KUKA KRL program: f1_Kuka_APT201T02S01.SRC

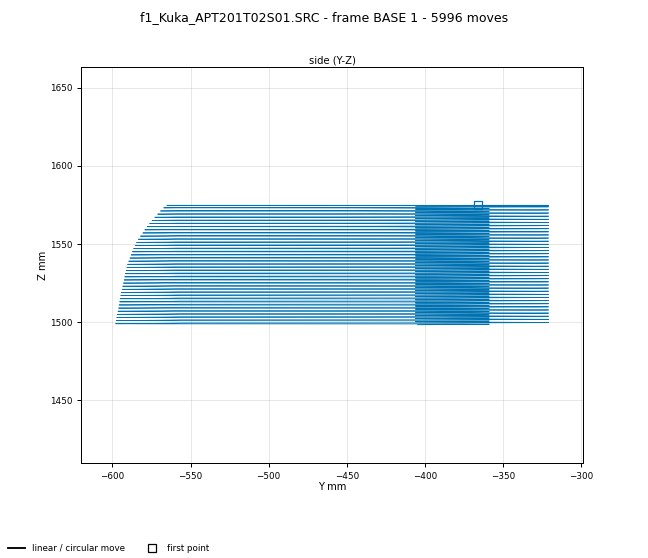
[picture p0: tool path of f1_Kuka_APT201T02S01.SRC in frame BASE 1, 5996 of 5998 moves have a stored position in this frame; points joined in program order, loops and branches not executed]
&ACCESS RVP
&REL 2
&PARAM TEMPLATE = C:\KRC\Roboter\Template\vorgabe
&PARAM EDITMASK = *
DEF f1_Kuka_APT201T02S01()


;FOLD INI;%{PE}%V3.2.0,%MKUKATPBASIS,%CINIT,%VCOMMON,%P
  ;FOLD BAS INI;%{E}%V3.2.0,%MKUKATPBASIS,%CINIT,%VINIT,%P
    GLOBAL INTERRUPT DECL 3 WHEN $STOPMESS==TRUE DO IR_STOPM ( )
    INTERRUPT ON 3
    BAS (#INITMOV,0 )
  ;ENDFOLD (BAS INI)
  ;FOLD USER INI;%{E}%V3.2.0,%MKUKATPUSER,%CINIT,%VINIT,%P
    ;Make your modifications here
  ;ENDFOLD (USER INI)
;ENDFOLD (INI)



;*** Make Initial Position Move
;FOLD PTP PPI1  Vel= 100 % PDAT1 Tool[0] Base[0];%{PE}%R 5.2.22,%MKUKATPBASIS,%CMOVE,%VPTP,%P 1:PTP, 2:PPI1, 3:, 5:100, 7:PDAT1
  $BWDSTART = FALSE
  PDAT_ACT = PPDAT1
  FDAT_ACT = FPPI1
  BAS(#PTP_PARAMS,100)
  PTP XPPI1
;ENDFOLD


;*** Auto Load the Correct TOOL and OFFSET
  ToolChange(2,1)


;*** Make Initial Position Move
;FOLD PTP PPI1  Vel= 100 % PDAT1 Tool[0] Base[0];%{PE}%R 5.2.22,%MKUKATPBASIS,%CMOVE,%VPTP,%P 1:PTP, 2:PPI1, 3:, 5:100, 7:PDAT1
  $BWDSTART = FALSE
  PDAT_ACT = PPDAT1
  FDAT_ACT = FPPI1
  BAS(#PTP_PARAMS,100)
  PTP XPPI1
;ENDFOLD

;*** Auto Load The Correct TOOL Data
  $tool=tool_data[2]

;*** Auto Load The Correct BASE Data
  $base=base_data[1]

  $ADVANCE = 5

SetRPM(8000)

MMPM(30000.0)
LIN {X 0.000,Y -365.799,Z 1574.800,A 0.000,B 0.000,C 90.000,E1 360.000} C_DIS
MMPM(15000.0)
LIN {X 0.000,Y -360.799,Z 1574.800,A 0.000,B 0.000,C 90.000,E1 360.000} C_DIS
MMPM(30000.0)
LIN {X -0.053,Y -359.426,Z 1574.800,A 0.000,B 0.000,C 90.000,E1 354.546} C_DIS
LIN {X 0.070,Y -358.890,Z 1574.800,A 0.000,B 0.000,C 90.000,E1 352.648} C_DIS
LIN {X -0.020,Y -359.563,Z 1574.800,A 0.000,B 0.000,C 90.000,E1 346.645} C_DIS
LIN {X 0.001,Y -361.801,Z 1574.800,A 0.000,B 0.000,C 90.000,E1 339.135} C_DIS
LIN {X -0.154,Y -362.053,Z 1574.800,A 0.000,B 0.000,C 90.000,E1 338.411} C_DIS
LIN {X 0.188,Y -365.979,Z 1574.800,A 0.000,B 0.000,C 90.000,E1 331.641} C_DIS
LIN {X 0.029,Y -366.387,Z 1574.800,A 0.000,B 0.000,C 90.000,E1 330.923} C_DIS
LIN {X -0.031,Y -371.355,Z 1574.800,A 0.000,B 0.000,C 90.000,E1 324.642} C_DIS
LIN {X -0.043,Y -371.766,Z 1574.800,A 0.000,B 0.000,C 90.000,E1 324.276} C_DIS
LIN {X 0.013,Y -377.358,Z 1574.800,A 0.000,B 0.000,C 90.000,E1 318.038} C_DIS
LIN {X 0.012,Y -378.235,Z 1574.800,A 0.000,B 0.000,C 90.000,E1 317.310} C_DIS
LIN {X 0.002,Y -383.940,Z 1574.800,A 0.000,B 0.000,C 90.000,E1 311.515} C_DIS
LIN {X 0.088,Y -384.893,Z 1574.800,A 0.000,B 0.000,C 90.000,E1 310.782} C_DIS
LIN {X 0.262,Y -390.610,Z 1574.800,A 0.000,B 0.000,C 90.000,E1 305.025} C_DIS
LIN {X 0.106,Y -391.104,Z 1574.800,A 0.000,B 0.000,C 90.000,E1 304.692} C_DIS
LIN {X 0.022,Y -391.648,Z 1574.800,A 0.000,B 0.000,C 90.000,E1 303.992} C_DIS
LIN {X -0.080,Y -396.825,Z 1574.800,A 0.000,B 0.000,C 90.000,E1 298.693} C_DIS
LIN {X -0.210,Y -397.120,Z 1574.800,A 0.000,B 0.000,C 90.000,E1 298.359} C_DIS
LIN {X -0.055,Y -401.597,Z 1574.800,A 0.000,B 0.000,C 90.000,E1 292.717} C_DIS
LIN {X 0.221,Y -404.659,Z 1574.800,A 0.000,B 0.000,C 90.000,E1 287.094} C_DIS
LIN {X -0.079,Y -404.735,Z 1574.800,A 0.000,B 0.000,C 90.000,E1 286.441} C_DIS
LIN {X 0.214,Y -406.099,Z 1574.800,A 0.000,B 0.000,C 90.000,E1 281.535} C_DIS
LIN {X -0.176,Y -406.094,Z 1574.800,A 0.000,B 0.000,C 90.000,E1 281.243} C_DIS
LIN {X -0.098,Y -405.680,Z 1574.800,A 0.000,B 0.000,C 90.000,E1 276.024} C_DIS
LIN {X -0.165,Y -405.058,Z 1574.800,A 0.000,B 0.000,C 90.000,E1 274.992} C_DIS
LIN {X -0.060,Y -403.497,Z 1574.800,A 0.000,B 0.000,C 90.000,E1 270.802} C_DIS
LIN {X -0.092,Y -403.288,Z 1574.800,A 0.000,B 0.000,C 90.000,E1 270.458} C_DIS
LIN {X 0.091,Y -398.931,Z 1574.800,A 0.000,B 0.000,C 90.000,E1 264.837} C_DIS
LIN {X -0.040,Y -393.108,Z 1574.800,A 0.000,B 0.000,C 90.000,E1 259.567} C_DIS
LIN {X -0.080,Y -392.836,Z 1574.800,A 0.000,B 0.000,C 90.000,E1 259.218} C_DIS
LIN {X 0.034,Y -385.993,Z 1574.800,A 0.000,B 0.000,C 90.000,E1 254.212} C_DIS
LIN {X -0.026,Y -385.267,Z 1574.800,A 0.000,B 0.000,C 90.000,E1 253.504} C_DIS
LIN {X -0.004,Y -384.767,Z 1574.800,A 0.000,B 0.000,C 90.000,E1 253.142} C_DIS
LIN {X 0.220,Y -377.972,Z 1574.800,A 0.000,B 0.000,C 90.000,E1 248.773} C_DIS
LIN {X -0.044,Y -376.233,Z 1574.800,A 0.000,B 0.000,C 90.000,E1 247.358} C_DIS
LIN {X 0.057,Y -374.944,Z 1574.800,A 0.000,B 0.000,C 90.000,E1 246.613} C_DIS
LIN {X -0.208,Y -368.417,Z 1574.800,A 0.000,B 0.000,C 90.000,E1 242.615} C_DIS
LIN {X 0.097,Y -366.047,Z 1574.800,A 0.000,B 0.000,C 90.000,E1 240.717} C_DIS
LIN {X 0.004,Y -359.196,Z 1574.800,A 0.000,B 0.000,C 90.000,E1 236.628} C_DIS
LIN {X 0.021,Y -355.842,Z 1574.800,A 0.000,B 0.000,C 90.000,E1 233.989} C_DIS
LIN {X -0.173,Y -348.793,Z 1574.800,A 0.000,B 0.000,C 90.000,E1 229.461} C_DIS
LIN {X -0.097,Y -346.185,Z 1574.800,A 0.000,B 0.000,C 90.000,E1 227.148} C_DIS
LIN {X -0.089,Y -345.065,Z 1574.800,A 0.000,B 0.000,C 90.000,E1 226.377} C_DIS
LIN {X 0.094,Y -338.586,Z 1574.800,A 0.000,B 0.000,C 90.000,E1 221.310} C_DIS
LIN {X 0.094,Y -336.840,Z 1574.800,A 0.000,B 0.000,C 90.000,E1 219.358} C_DIS
LIN {X 0.014,Y -330.861,Z 1574.800,A 0.000,B 0.000,C 90.000,E1 213.865} C_DIS
LIN {X 0.149,Y -329.296,Z 1574.800,A 0.000,B 0.000,C 90.000,E1 211.465} C_DIS
LIN {X -0.154,Y -324.669,Z 1574.800,A 0.000,B 0.000,C 90.000,E1 205.540} C_DIS
LIN {X 0.174,Y -323.838,Z 1574.800,A 0.000,B 0.000,C 90.000,E1 203.078} C_DIS
LIN {X -0.018,Y -321.123,Z 1574.800,A 0.000,B 0.000,C 90.000,E1 194.662} C_DIS
LIN {X 0.138,Y -320.932,Z 1574.800,A 0.000,B 0.000,C 90.000,E1 193.828} C_DIS
LIN {X -0.076,Y -321.563,Z 1574.800,A 0.000,B 0.000,C 90.000,E1 185.796} C_DIS
LIN {X -0.143,Y -324.415,Z 1574.800,A 0.000,B 0.000,C 90.000,E1 178.165} C_DIS
LIN {X -0.141,Y -325.376,Z 1574.800,A 0.000,B 0.000,C 90.000,E1 176.963} C_DIS
LIN {X -0.100,Y -329.112,Z 1574.800,A 0.000,B 0.000,C 90.000,E1 170.971} C_DIS
LIN {X 0.061,Y -334.260,Z 1574.800,A 0.000,B 0.000,C 90.000,E1 166.589} C_DIS
LIN {X 0.067,Y -335.488,Z 1574.800,A 0.000,B 0.000,C 90.000,E1 165.408} C_DIS
LIN {X 0.143,Y -340.932,Z 1574.800,A 0.000,B 0.000,C 90.000,E1 161.094} C_DIS
LIN {X -0.172,Y -342.138,Z 1574.800,A 0.000,B 0.000,C 90.000,E1 160.369} C_DIS
LIN {X -0.058,Y -347.939,Z 1574.800,A 0.000,B 0.000,C 90.000,E1 156.102} C_DIS
LIN {X -0.082,Y -354.260,Z 1574.800,A 0.000,B 0.000,C 90.000,E1 152.666} C_DIS
LIN {X -0.222,Y -361.406,Z 1574.800,A 0.000,B 0.000,C 90.000,E1 148.535} C_DIS
LIN {X 0.064,Y -368.758,Z 1574.800,A 0.000,B 0.000,C 90.000,E1 145.135} C_DIS
LIN {X 0.064,Y -377.030,Z 1574.800,A 0.000,B 0.000,C 90.000,E1 141.090} C_DIS
LIN {X -0.061,Y -383.435,Z 1574.800,A 0.000,B 0.000,C 90.000,E1 138.566} C_DIS
LIN {X -0.015,Y -385.037,Z 1574.800,A 0.000,B 0.000,C 90.000,E1 137.838} C_DIS
LIN {X -0.004,Y -394.325,Z 1574.800,A 0.000,B 0.000,C 90.000,E1 133.905} C_DIS
LIN {X 0.107,Y -399.276,Z 1574.800,A 0.000,B 0.000,C 90.000,E1 132.123} C_DIS
LIN {X 0.210,Y -400.192,Z 1574.800,A 0.000,B 0.000,C 90.000,E1 131.757} C_DIS
LIN {X -0.113,Y -409.687,Z 1574.800,A 0.000,B 0.000,C 90.000,E1 127.971} C_DIS
LIN {X 0.046,Y -415.746,Z 1574.800,A 0.000,B 0.000,C 90.000,E1 125.884} C_DIS
LIN {X 0.152,Y -425.188,Z 1574.800,A 0.000,B 0.000,C 90.000,E1 122.133} C_DIS
LIN {X 0.086,Y -430.187,Z 1574.800,A 0.000,B 0.000,C 90.000,E1 120.463} C_DIS
LIN {X 0.085,Y -431.108,Z 1574.800,A 0.000,B 0.000,C 90.000,E1 120.129} C_DIS
LIN {X 0.032,Y -440.206,Z 1574.800,A 0.000,B 0.000,C 90.000,E1 116.488} C_DIS
LIN {X 0.039,Y -444.962,Z 1574.800,A 0.000,B 0.000,C 90.000,E1 114.847} C_DIS
LIN {X -0.108,Y -454.089,Z 1574.800,A 0.000,B 0.000,C 90.000,E1 110.972} C_DIS
LIN {X 0.003,Y -456.743,Z 1574.800,A 0.000,B 0.000,C 90.000,E1 109.993} C_DIS
LIN {X -0.096,Y -457.517,Z 1574.800,A 0.000,B 0.000,C 90.000,E1 109.685} C_DIS
LIN {X -0.150,Y -466.200,Z 1574.800,A 0.000,B 0.000,C 90.000,E1 105.552} C_DIS
LIN {X 0.026,Y -467.764,Z 1574.800,A 0.000,B 0.000,C 90.000,E1 104.898} C_DIS
LIN {X -0.209,Y -469.313,Z 1574.800,A 0.000,B 0.000,C 90.000,E1 103.883} C_DIS
LIN {X 0.252,Y -548.916,Z 1574.800,A 0.000,B 0.000,C 90.000,E1 103.828} C_DIS
LIN {X -0.055,Y -550.377,Z 1574.800,A 0.000,B 0.000,C 90.000,E1 103.647} C_DIS
LIN {X 0.049,Y -551.250,Z 1574.800,A 0.000,B 0.000,C 90.000,E1 103.355} C_DIS
LIN {X -0.263,Y -552.432,Z 1574.800,A 0.000,B 0.000,C 90.000,E1 102.827} C_DIS
LIN {X 0.096,Y -553.523,Z 1574.800,A 0.000,B 0.000,C 90.000,E1 101.951} C_DIS
LIN {X -0.073,Y -554.401,Z 1574.800,A 0.000,B 0.000,C 90.000,E1 101.130} C_DIS
LIN {X -0.236,Y -555.112,Z 1574.800,A 0.000,B 0.000,C 90.000,E1 100.310} C_DIS
LIN {X -0.102,Y -556.191,Z 1574.800,A 0.000,B 0.000,C 90.000,E1 98.624} C_DIS
LIN {X -0.289,Y -556.849,Z 1574.800,A 0.000,B 0.000,C 90.000,E1 97.530} C_DIS
LIN {X -0.203,Y -557.535,Z 1574.800,A 0.000,B 0.000,C 90.000,E1 95.853} C_DIS
LIN {X -0.219,Y -557.914,Z 1574.800,A 0.000,B 0.000,C 90.000,E1 94.188} C_DIS
LIN {X -0.221,Y -558.368,Z 1574.800,A 0.000,B 0.000,C 90.000,E1 92.522} C_DIS
LIN {X 0.226,Y -558.750,Z 1574.800,A 0.000,B 0.000,C 90.000,E1 91.088} C_DIS
LIN {X -0.272,Y -559.196,Z 1574.800,A 0.000,B 0.000,C 90.000,E1 89.198} C_DIS
LIN {X -0.191,Y -559.752,Z 1574.800,A 0.000,B 0.000,C 90.000,E1 87.249} C_DIS
LIN {X -0.157,Y -560.343,Z 1574.800,A 0.000,B 0.000,C 90.000,E1 85.584} C_DIS
LIN {X 0.022,Y -561.145,Z 1574.800,A 0.000,B 0.000,C 90.000,E1 83.628} C_DIS
LIN {X -0.132,Y -562.271,Z 1574.800,A 0.000,B 0.000,C 90.000,E1 81.432} C_DIS
LIN {X -0.235,Y -563.276,Z 1574.800,A 0.000,B 0.000,C 90.000,E1 79.511} C_DIS
LIN {X 0.073,Y -564.218,Z 1574.800,A 0.000,B 0.000,C 90.000,E1 77.825} C_DIS
LIN {X 0.080,Y -564.877,Z 1574.800,A 0.000,B 0.000,C 90.000,E1 76.172} C_DIS
LIN {X -0.219,Y -565.104,Z 1574.800,A 0.000,B 0.000,C 90.000,E1 75.102} C_DIS
LIN {X -0.128,Y -565.147,Z 1574.800,A 0.000,B 0.000,C 90.000,E1 74.267} C_DIS
LIN {X 0.121,Y -564.945,Z 1574.800,A 0.000,B 0.000,C 90.000,E1 73.142} C_DIS
LIN {X 0.053,Y -564.549,Z 1574.800,A 0.000,B 0.000,C 90.000,E1 72.598} C_DIS
LIN {X -0.014,Y -563.765,Z 1574.800,A 0.000,B 0.000,C 90.000,E1 72.054} C_DIS
LIN {X -0.167,Y -562.900,Z 1574.800,A 0.000,B 0.000,C 90.000,E1 71.764} C_DIS
LIN {X -0.031,Y -562.209,Z 1574.800,A 0.000,B 0.000,C 90.000,E1 71.638} C_DIS
LIN {X -0.274,Y -561.841,Z 1574.800,A 0.000,B 0.000,C 90.000,E1 71.638} C_DIS
LIN {X 0.177,Y -473.244,Z 1574.800,A 0.000,B 0.000,C 90.000,E1 71.583} C_DIS
LIN {X 0.025,Y -465.713,Z 1574.800,A 0.000,B 0.000,C 90.000,E1 67.102} C_DIS
LIN {X -0.179,Y -456.183,Z 1574.800,A 0.000,B 0.000,C 90.000,E1 62.359} C_DIS
LIN {X -0.073,Y -455.666,Z 1574.800,A 0.000,B 0.000,C 90.000,E1 62.025} C_DIS
LIN {X -0.081,Y -454.178,Z 1574.800,A 0.000,B 0.000,C 90.000,E1 61.385} C_DIS
LIN {X 0.021,Y -445.148,Z 1574.800,A 0.000,B 0.000,C 90.000,E1 57.168} C_DIS
LIN {X 0.146,Y -443.995,Z 1574.800,A 0.000,B 0.000,C 90.000,E1 56.501} C_DIS
LIN {X 0.091,Y -433.537,Z 1574.800,A 0.000,B 0.000,C 90.000,E1 51.904} C_DIS
LIN {X -0.063,Y -431.699,Z 1574.800,A 0.000,B 0.000,C 90.000,E1 50.928} C_DIS
LIN {X 0.096,Y -429.255,Z 1574.800,A 0.000,B 0.000,C 90.000,E1 49.908} C_DIS
LIN {X -0.126,Y -419.923,Z 1574.800,A 0.000,B 0.000,C 90.000,E1 45.567} C_DIS
LIN {X -0.048,Y -418.732,Z 1574.800,A 0.000,B 0.000,C 90.000,E1 44.879} C_DIS
LIN {X -0.082,Y -409.803,Z 1574.800,A 0.000,B 0.000,C 90.000,E1 40.782} C_DIS
LIN {X -0.045,Y -406.207,Z 1574.800,A 0.000,B 0.000,C 90.000,E1 38.705} C_DIS
LIN {X 0.100,Y -405.567,Z 1574.800,A 0.000,B 0.000,C 90.000,E1 38.338} C_DIS
LIN {X 0.175,Y -396.741,Z 1574.800,A 0.000,B 0.000,C 90.000,E1 33.785} C_DIS
LIN {X 0.155,Y -393.529,Z 1574.800,A 0.000,B 0.000,C 90.000,E1 31.671} C_DIS
LIN {X -0.093,Y -386.172,Z 1574.800,A 0.000,B 0.000,C 90.000,E1 27.436} C_DIS
LIN {X 0.055,Y -382.972,Z 1574.800,A 0.000,B 0.000,C 90.000,E1 24.899} C_DIS
LIN {X 0.036,Y -376.689,Z 1574.800,A 0.000,B 0.000,C 90.000,E1 20.556} C_DIS
LIN {X 0.019,Y -373.753,Z 1574.800,A 0.000,B 0.000,C 90.000,E1 17.638} C_DIS
LIN {X -0.034,Y -372.850,Z 1574.800,A 0.000,B 0.000,C 90.000,E1 16.913} C_DIS
LIN {X -0.131,Y -367.590,Z 1574.800,A 0.000,B 0.000,C 90.000,E1 11.771} C_DIS
LIN {X -0.047,Y -366.471,Z 1574.800,A 0.000,B 0.000,C 90.000,E1 9.905} C_DIS
LIN {X -0.109,Y -361.776,Z 1574.800,A 0.000,B 0.000,C 90.000,E1 3.955} C_DIS
LIN {X 0.136,Y -360.896,Z 1574.800,A 0.000,B 0.000,C 90.000,E1 0.172} C_DIS
LIN {X -0.053,Y -359.426,Z 1574.770,A 0.000,B 0.000,C 90.000,E1 354.546} C_DIS
LIN {X 0.070,Y -358.890,Z 1574.759,A 0.000,B 0.000,C 90.000,E1 352.648} C_DIS
LIN {X -0.020,Y -359.563,Z 1574.726,A 0.000,B 0.000,C 90.000,E1 346.645} C_DIS
LIN {X 0.001,Y -361.801,Z 1574.684,A 0.000,B 0.000,C 90.000,E1 339.135} C_DIS
LIN {X -0.154,Y -362.053,Z 1574.680,A 0.000,B 0.000,C 90.000,E1 338.411} C_DIS
LIN {X 0.189,Y -365.980,Z 1574.643,A 0.000,B 0.000,C 90.000,E1 331.641} C_DIS
LIN {X 0.029,Y -366.387,Z 1574.639,A 0.000,B 0.000,C 90.000,E1 330.923} C_DIS
LIN {X -0.031,Y -371.355,Z 1574.604,A 0.000,B 0.000,C 90.000,E1 324.642} C_DIS
LIN {X -0.043,Y -371.766,Z 1574.602,A 0.000,B 0.000,C 90.000,E1 324.276} C_DIS
LIN {X 0.013,Y -377.358,Z 1574.567,A 0.000,B 0.000,C 90.000,E1 318.038} C_DIS
LIN {X 0.012,Y -378.235,Z 1574.563,A 0.000,B 0.000,C 90.000,E1 317.310} C_DIS
LIN {X 0.002,Y -383.940,Z 1574.531,A 0.000,B 0.000,C 90.000,E1 311.515} C_DIS
LIN {X 0.088,Y -384.893,Z 1574.527,A 0.000,B 0.000,C 90.000,E1 310.782} C_DIS
LIN {X 0.262,Y -390.610,Z 1574.495,A 0.000,B 0.000,C 90.000,E1 305.025} C_DIS
LIN {X 0.106,Y -391.104,Z 1574.493,A 0.000,B 0.000,C 90.000,E1 304.692} C_DIS
LIN {X 0.022,Y -391.648,Z 1574.489,A 0.000,B 0.000,C 90.000,E1 303.992} C_DIS
LIN {X -0.080,Y -396.825,Z 1574.459,A 0.000,B 0.000,C 90.000,E1 298.693} C_DIS
LIN {X -0.210,Y -397.120,Z 1574.457,A 0.000,B 0.000,C 90.000,E1 298.359} C_DIS
LIN {X -0.055,Y -401.597,Z 1574.426,A 0.000,B 0.000,C 90.000,E1 292.717} C_DIS
LIN {X 0.222,Y -404.659,Z 1574.395,A 0.000,B 0.000,C 90.000,E1 287.094} C_DIS
LIN {X -0.079,Y -404.735,Z 1574.391,A 0.000,B 0.000,C 90.000,E1 286.441} C_DIS
LIN {X 0.214,Y -406.099,Z 1574.364,A 0.000,B 0.000,C 90.000,E1 281.535} C_DIS
LIN {X -0.176,Y -406.094,Z 1574.362,A 0.000,B 0.000,C 90.000,E1 281.243} C_DIS
LIN {X -0.097,Y -405.680,Z 1574.333,A 0.000,B 0.000,C 90.000,E1 276.024} C_DIS
LIN {X -0.165,Y -405.058,Z 1574.328,A 0.000,B 0.000,C 90.000,E1 274.992} C_DIS
LIN {X -0.060,Y -403.497,Z 1574.304,A 0.000,B 0.000,C 90.000,E1 270.802} C_DIS
LIN {X -0.092,Y -403.288,Z 1574.302,A 0.000,B 0.000,C 90.000,E1 270.458} C_DIS
LIN {X 0.091,Y -398.931,Z 1574.271,A 0.000,B 0.000,C 90.000,E1 264.837} C_DIS
LIN {X -0.040,Y -393.108,Z 1574.242,A 0.000,B 0.000,C 90.000,E1 259.567} C_DIS
LIN {X -0.079,Y -392.835,Z 1574.240,A 0.000,B 0.000,C 90.000,E1 259.218} C_DIS
LIN {X 0.034,Y -385.993,Z 1574.212,A 0.000,B 0.000,C 90.000,E1 254.212} C_DIS
LIN {X -0.026,Y -385.267,Z 1574.208,A 0.000,B 0.000,C 90.000,E1 253.504} C_DIS
LIN {X -0.004,Y -384.768,Z 1574.206,A 0.000,B 0.000,C 90.000,E1 253.142} C_DIS
LIN {X 0.221,Y -377.973,Z 1574.182,A 0.000,B 0.000,C 90.000,E1 248.773} C_DIS
LIN {X -0.044,Y -376.233,Z 1574.174,A 0.000,B 0.000,C 90.000,E1 247.358} C_DIS
LIN {X 0.057,Y -374.944,Z 1574.170,A 0.000,B 0.000,C 90.000,E1 246.613} C_DIS
LIN {X -0.208,Y -368.417,Z 1574.148,A 0.000,B 0.000,C 90.000,E1 242.615} C_DIS
LIN {X 0.097,Y -366.047,Z 1574.137,A 0.000,B 0.000,C 90.000,E1 240.717} C_DIS
LIN {X 0.004,Y -359.196,Z 1574.115,A 0.000,B 0.000,C 90.000,E1 236.628} C_DIS
LIN {X 0.021,Y -355.842,Z 1574.100,A 0.000,B 0.000,C 90.000,E1 233.989} C_DIS
LIN {X -0.173,Y -348.793,Z 1574.075,A 0.000,B 0.000,C 90.000,E1 229.461} C_DIS
LIN {X -0.097,Y -346.185,Z 1574.062,A 0.000,B 0.000,C 90.000,E1 227.148} C_DIS
LIN {X -0.088,Y -345.065,Z 1574.058,A 0.000,B 0.000,C 90.000,E1 226.377} C_DIS
LIN {X 0.094,Y -338.586,Z 1574.030,A 0.000,B 0.000,C 90.000,E1 221.310} C_DIS
LIN {X 0.094,Y -336.840,Z 1574.019,A 0.000,B 0.000,C 90.000,E1 219.358} C_DIS
LIN {X 0.014,Y -330.861,Z 1573.988,A 0.000,B 0.000,C 90.000,E1 213.865} C_DIS
LIN {X 0.149,Y -329.296,Z 1573.975,A 0.000,B 0.000,C 90.000,E1 211.465} C_DIS
LIN {X -0.154,Y -324.669,Z 1573.942,A 0.000,B 0.000,C 90.000,E1 205.540} C_DIS
LIN {X 0.174,Y -323.837,Z 1573.928,A 0.000,B 0.000,C 90.000,E1 203.078} C_DIS
LIN {X -0.017,Y -321.124,Z 1573.881,A 0.000,B 0.000,C 90.000,E1 194.662} C_DIS
LIN {X 0.138,Y -320.932,Z 1573.877,A 0.000,B 0.000,C 90.000,E1 193.828} C_DIS
LIN {X -0.076,Y -321.562,Z 1573.832,A 0.000,B 0.000,C 90.000,E1 185.796} C_DIS
LIN {X -0.143,Y -324.415,Z 1573.790,A 0.000,B 0.000,C 90.000,E1 178.165} C_DIS
LIN {X -0.141,Y -325.376,Z 1573.783,A 0.000,B 0.000,C 90.000,E1 176.963} C_DIS
LIN {X -0.100,Y -329.112,Z 1573.750,A 0.000,B 0.000,C 90.000,E1 170.971} C_DIS
LIN {X 0.061,Y -334.260,Z 1573.726,A 0.000,B 0.000,C 90.000,E1 166.589} C_DIS
LIN {X 0.067,Y -335.488,Z 1573.719,A 0.000,B 0.000,C 90.000,E1 165.408} C_DIS
LIN {X 0.143,Y -340.932,Z 1573.695,A 0.000,B 0.000,C 90.000,E1 161.094} C_DIS
LIN {X -0.172,Y -342.138,Z 1573.691,A 0.000,B 0.000,C 90.000,E1 160.369} C_DIS
LIN {X -0.058,Y -347.939,Z 1573.667,A 0.000,B 0.000,C 90.000,E1 156.102} C_DIS
LIN {X -0.081,Y -354.259,Z 1573.648,A 0.000,B 0.000,C 90.000,E1 152.666} C_DIS
LIN {X -0.222,Y -361.406,Z 1573.625,A 0.000,B 0.000,C 90.000,E1 148.535} C_DIS
LIN {X 0.065,Y -368.758,Z 1573.606,A 0.000,B 0.000,C 90.000,E1 145.135} C_DIS
LIN {X 0.065,Y -377.029,Z 1573.584,A 0.000,B 0.000,C 90.000,E1 141.090} C_DIS
LIN {X -0.061,Y -383.435,Z 1573.570,A 0.000,B 0.000,C 90.000,E1 138.566} C_DIS
LIN {X -0.015,Y -385.037,Z 1573.566,A 0.000,B 0.000,C 90.000,E1 137.838} C_DIS
LIN {X -0.004,Y -394.325,Z 1573.544,A 0.000,B 0.000,C 90.000,E1 133.905} C_DIS
LIN {X 0.107,Y -399.276,Z 1573.534,A 0.000,B 0.000,C 90.000,E1 132.123} C_DIS
LIN {X 0.210,Y -400.192,Z 1573.532,A 0.000,B 0.000,C 90.000,E1 131.757} C_DIS
LIN {X -0.113,Y -409.687,Z 1573.511,A 0.000,B 0.000,C 90.000,E1 127.971} C_DIS
LIN {X 0.046,Y -415.746,Z 1573.499,A 0.000,B 0.000,C 90.000,E1 125.884} C_DIS
LIN {X 0.153,Y -425.188,Z 1573.479,A 0.000,B 0.000,C 90.000,E1 122.133} C_DIS
LIN {X 0.087,Y -430.186,Z 1573.469,A 0.000,B 0.000,C 90.000,E1 120.463} C_DIS
LIN {X 0.086,Y -431.107,Z 1573.468,A 0.000,B 0.000,C 90.000,E1 120.129} C_DIS
LIN {X 0.032,Y -440.207,Z 1573.447,A 0.000,B 0.000,C 90.000,E1 116.488} C_DIS
LIN {X 0.039,Y -444.962,Z 1573.438,A 0.000,B 0.000,C 90.000,E1 114.847} C_DIS
LIN {X -0.108,Y -454.089,Z 1573.417,A 0.000,B 0.000,C 90.000,E1 110.972} C_DIS
LIN {X 0.005,Y -456.742,Z 1573.411,A 0.000,B 0.000,C 90.000,E1 109.993} C_DIS
LIN {X -0.096,Y -457.517,Z 1573.409,A 0.000,B 0.000,C 90.000,E1 109.685} C_DIS
LIN {X -0.047,Y -465.767,Z 1573.387,A 0.000,B 0.000,C 90.000,E1 105.717} C_DIS
LIN {X -0.088,Y -548.675,Z 1573.387,A 0.000,B 0.000,C 90.000,E1 105.717} C_DIS
LIN {X -0.153,Y -548.982,Z 1573.387,A 0.000,B 0.000,C 90.000,E1 105.717} C_DIS
LIN {X -0.177,Y -550.294,Z 1573.386,A 0.000,B 0.000,C 90.000,E1 105.552} C_DIS
LIN {X 0.069,Y -551.293,Z 1573.385,A 0.000,B 0.000,C 90.000,E1 105.245} C_DIS
LIN {X 0.175,Y -551.975,Z 1573.383,A 0.000,B 0.000,C 90.000,E1 104.954} C_DIS
LIN {X 0.004,Y -552.984,Z 1573.380,A 0.000,B 0.000,C 90.000,E1 104.411} C_DIS
LIN {X 0.239,Y -553.715,Z 1573.377,A 0.000,B 0.000,C 90.000,E1 103.828} C_DIS
LIN {X 0.196,Y -554.850,Z 1573.371,A 0.000,B 0.000,C 90.000,E1 102.715} C_DIS
LIN {X -0.236,Y -555.849,Z 1573.363,A 0.000,B 0.000,C 90.000,E1 101.366} C_DIS
LIN {X -0.248,Y -556.511,Z 1573.357,A 0.000,B 0.000,C 90.000,E1 100.254} C_DIS
LIN {X 0.051,Y -557.419,Z 1573.346,A 0.000,B 0.000,C 90.000,E1 98.276} C_DIS
LIN {X -0.181,Y -557.796,Z 1573.341,A 0.000,B 0.000,C 90.000,E1 97.466} C_DIS
LIN {X -0.147,Y -558.339,Z 1573.332,A 0.000,B 0.000,C 90.000,E1 95.796} C_DIS
LIN {X -0.143,Y -558.609,Z 1573.323,A 0.000,B 0.000,C 90.000,E1 94.131} C_DIS
LIN {X -0.131,Y -558.995,Z 1573.314,A 0.000,B 0.000,C 90.000,E1 92.465} C_DIS
LIN {X -0.230,Y -559.336,Z 1573.306,A 0.000,B 0.000,C 90.000,E1 91.088} C_DIS
LIN {X -0.156,Y -559.756,Z 1573.295,A 0.000,B 0.000,C 90.000,E1 89.141} C_DIS
LIN {X -0.061,Y -560.327,Z 1573.284,A 0.000,B 0.000,C 90.000,E1 87.192} C_DIS
LIN {X -0.015,Y -560.941,Z 1573.275,A 0.000,B 0.000,C 90.000,E1 85.527} C_DIS
LIN {X 0.178,Y -561.807,Z 1573.264,A 0.000,B 0.000,C 90.000,E1 83.571} C_DIS
LIN {X 0.041,Y -563.034,Z 1573.252,A 0.000,B 0.000,C 90.000,E1 81.376} C_DIS
LIN {X -0.044,Y -564.180,Z 1573.241,A 0.000,B 0.000,C 90.000,E1 79.454} C_DIS
LIN {X -0.152,Y -565.281,Z 1573.232,A 0.000,B 0.000,C 90.000,E1 77.813} C_DIS
LIN {X -0.241,Y -566.169,Z 1573.223,A 0.000,B 0.000,C 90.000,E1 76.172} C_DIS
LIN {X 0.192,Y -566.734,Z 1573.215,A 0.000,B 0.000,C 90.000,E1 74.755} C_DIS
LIN {X 0.240,Y -567.099,Z 1573.208,A 0.000,B 0.000,C 90.000,E1 73.378} C_DIS
LIN {X -0.193,Y -567.140,Z 1573.203,A 0.000,B 0.000,C 90.000,E1 72.598} C_DIS
LIN {X 0.244,Y -566.843,Z 1573.197,A 0.000,B 0.000,C 90.000,E1 71.456} C_DIS
LIN {X -0.198,Y -566.323,Z 1573.193,A 0.000,B 0.000,C 90.000,E1 70.678} C_DIS
LIN {X -0.065,Y -565.425,Z 1573.190,A 0.000,B 0.000,C 90.000,E1 70.115} C_DIS
LIN {X -0.069,Y -564.450,Z 1573.188,A 0.000,B 0.000,C 90.000,E1 69.752} C_DIS
LIN {X 0.067,Y -563.822,Z 1573.187,A 0.000,B 0.000,C 90.000,E1 69.625} C_DIS
LIN {X 0.239,Y -563.373,Z 1573.187,A 0.000,B 0.000,C 90.000,E1 69.571} C_DIS
LIN {X 0.182,Y -563.196,Z 1573.187,A 0.000,B 0.000,C 90.000,E1 69.571} C_DIS
LIN {X 0.104,Y -469.466,Z 1573.187,A 0.000,B 0.000,C 90.000,E1 69.571} C_DIS
LIN {X -0.082,Y -465.606,Z 1573.172,A 0.000,B 0.000,C 90.000,E1 67.050} C_DIS
LIN {X -0.203,Y -456.601,Z 1573.148,A 0.000,B 0.000,C 90.000,E1 62.615} C_DIS
LIN {X -0.203,Y -455.561,Z 1573.144,A 0.000,B 0.000,C 90.000,E1 61.975} C_DIS
LIN {X -0.199,Y -445.620,Z 1573.119,A 0.000,B 0.000,C 90.000,E1 57.454} C_DIS
LIN {X 0.233,Y -443.853,Z 1573.114,A 0.000,B 0.000,C 90.000,E1 56.421} C_DIS
LIN {X 0.245,Y -434.703,Z 1573.092,A 0.000,B 0.000,C 90.000,E1 52.477} C_DIS
LIN {X -0.252,Y -431.576,Z 1573.083,A 0.000,B 0.000,C 90.000,E1 50.884} C_DIS
LIN {X -0.044,Y -421.692,Z 1573.058,A 0.000,B 0.000,C 90.000,E1 46.500} C_DIS
LIN {X 0.025,Y -418.597,Z 1573.049,A 0.000,B 0.000,C 90.000,E1 44.798} C_DIS
LIN {X -0.170,Y -409.031,Z 1573.024,A 0.000,B 0.000,C 90.000,E1 40.378} C_DIS
LIN {X 0.012,Y -406.092,Z 1573.015,A 0.000,B 0.000,C 90.000,E1 38.624} C_DIS
LIN {X -0.131,Y -403.868,Z 1573.009,A 0.000,B 0.000,C 90.000,E1 37.604} C_DIS
LIN {X -0.038,Y -395.519,Z 1572.984,A 0.000,B 0.000,C 90.000,E1 33.038} C_DIS
LIN {X -0.218,Y -393.987,Z 1572.978,A 0.000,B 0.000,C 90.000,E1 32.005} C_DIS
LIN {X 0.051,Y -392.679,Z 1572.974,A 0.000,B 0.000,C 90.000,E1 31.258} C_DIS
LIN {X 0.092,Y -385.076,Z 1572.948,A 0.000,B 0.000,C 90.000,E1 26.616} C_DIS
LIN {X 0.060,Y -382.887,Z 1572.938,A 0.000,B 0.000,C 90.000,E1 24.823} C_DIS
LIN {X 0.007,Y -376.178,Z 1572.912,A 0.000,B 0.000,C 90.000,E1 20.120} C_DIS
LIN {X -0.124,Y -373.690,Z 1572.898,A 0.000,B 0.000,C 90.000,E1 17.583} C_DIS
LIN {X 0.011,Y -368.087,Z 1572.869,A 0.000,B 0.000,C 90.000,E1 12.411} C_DIS
LIN {X -0.181,Y -366.407,Z 1572.855,A 0.000,B 0.000,C 90.000,E1 9.849} C_DIS
LIN {X 0.118,Y -361.742,Z 1572.822,A 0.000,B 0.000,C 90.000,E1 3.841} C_DIS
LIN {X 0.004,Y -360.864,Z 1572.801,A 0.000,B 0.000,C 90.000,E1 0.115} C_DIS
LIN {X -0.053,Y -359.426,Z 1572.770,A 0.000,B 0.000,C 90.000,E1 354.546} C_DIS
LIN {X 0.070,Y -358.890,Z 1572.759,A 0.000,B 0.000,C 90.000,E1 352.648} C_DIS
LIN {X -0.020,Y -359.563,Z 1572.726,A 0.000,B 0.000,C 90.000,E1 346.645} C_DIS
LIN {X 0.001,Y -361.801,Z 1572.684,A 0.000,B 0.000,C 90.000,E1 339.135} C_DIS
LIN {X -0.154,Y -362.053,Z 1572.680,A 0.000,B 0.000,C 90.000,E1 338.411} C_DIS
LIN {X 0.189,Y -365.980,Z 1572.643,A 0.000,B 0.000,C 90.000,E1 331.641} C_DIS
LIN {X 0.029,Y -366.387,Z 1572.639,A 0.000,B 0.000,C 90.000,E1 330.923} C_DIS
LIN {X -0.031,Y -371.355,Z 1572.604,A 0.000,B 0.000,C 90.000,E1 324.642} C_DIS
LIN {X -0.043,Y -371.766,Z 1572.602,A 0.000,B 0.000,C 90.000,E1 324.276} C_DIS
LIN {X 0.013,Y -377.358,Z 1572.567,A 0.000,B 0.000,C 90.000,E1 318.038} C_DIS
LIN {X 0.012,Y -378.235,Z 1572.563,A 0.000,B 0.000,C 90.000,E1 317.310} C_DIS
LIN {X 0.002,Y -383.940,Z 1572.531,A 0.000,B 0.000,C 90.000,E1 311.515} C_DIS
LIN {X 0.088,Y -384.893,Z 1572.527,A 0.000,B 0.000,C 90.000,E1 310.782} C_DIS
LIN {X 0.262,Y -390.610,Z 1572.495,A 0.000,B 0.000,C 90.000,E1 305.025} C_DIS
LIN {X 0.106,Y -391.104,Z 1572.493,A 0.000,B 0.000,C 90.000,E1 304.692} C_DIS
LIN {X 0.022,Y -391.648,Z 1572.489,A 0.000,B 0.000,C 90.000,E1 303.992} C_DIS
LIN {X -0.080,Y -396.825,Z 1572.459,A 0.000,B 0.000,C 90.000,E1 298.693} C_DIS
LIN {X -0.210,Y -397.120,Z 1572.457,A 0.000,B 0.000,C 90.000,E1 298.359} C_DIS
LIN {X -0.055,Y -401.597,Z 1572.426,A 0.000,B 0.000,C 90.000,E1 292.717} C_DIS
LIN {X 0.222,Y -404.659,Z 1572.395,A 0.000,B 0.000,C 90.000,E1 287.094} C_DIS
LIN {X -0.079,Y -404.735,Z 1572.391,A 0.000,B 0.000,C 90.000,E1 286.441} C_DIS
LIN {X 0.214,Y -406.099,Z 1572.364,A 0.000,B 0.000,C 90.000,E1 281.535} C_DIS
LIN {X -0.176,Y -406.094,Z 1572.362,A 0.000,B 0.000,C 90.000,E1 281.243} C_DIS
LIN {X -0.097,Y -405.680,Z 1572.333,A 0.000,B 0.000,C 90.000,E1 276.024} C_DIS
LIN {X -0.165,Y -405.058,Z 1572.328,A 0.000,B 0.000,C 90.000,E1 274.992} C_DIS
LIN {X -0.060,Y -403.497,Z 1572.304,A 0.000,B 0.000,C 90.000,E1 270.802} C_DIS
LIN {X -0.092,Y -403.288,Z 1572.302,A 0.000,B 0.000,C 90.000,E1 270.458} C_DIS
LIN {X 0.091,Y -398.931,Z 1572.271,A 0.000,B 0.000,C 90.000,E1 264.837} C_DIS
LIN {X -0.040,Y -393.108,Z 1572.242,A 0.000,B 0.000,C 90.000,E1 259.567} C_DIS
LIN {X -0.079,Y -392.835,Z 1572.240,A 0.000,B 0.000,C 90.000,E1 259.218} C_DIS
LIN {X 0.034,Y -385.993,Z 1572.212,A 0.000,B 0.000,C 90.000,E1 254.212} C_DIS
LIN {X -0.026,Y -385.267,Z 1572.208,A 0.000,B 0.000,C 90.000,E1 253.504} C_DIS
LIN {X -0.004,Y -384.768,Z 1572.206,A 0.000,B 0.000,C 90.000,E1 253.142} C_DIS
LIN {X 0.221,Y -377.973,Z 1572.182,A 0.000,B 0.000,C 90.000,E1 248.773} C_DIS
LIN {X -0.044,Y -376.233,Z 1572.174,A 0.000,B 0.000,C 90.000,E1 247.358} C_DIS
LIN {X 0.057,Y -374.944,Z 1572.170,A 0.000,B 0.000,C 90.000,E1 246.613} C_DIS
LIN {X -0.208,Y -368.417,Z 1572.148,A 0.000,B 0.000,C 90.000,E1 242.615} C_DIS
LIN {X 0.097,Y -366.047,Z 1572.137,A 0.000,B 0.000,C 90.000,E1 240.717} C_DIS
LIN {X 0.004,Y -359.196,Z 1572.115,A 0.000,B 0.000,C 90.000,E1 236.628} C_DIS
LIN {X 0.021,Y -355.842,Z 1572.100,A 0.000,B 0.000,C 90.000,E1 233.989} C_DIS
LIN {X -0.173,Y -348.793,Z 1572.075,A 0.000,B 0.000,C 90.000,E1 229.461} C_DIS
LIN {X -0.097,Y -346.185,Z 1572.062,A 0.000,B 0.000,C 90.000,E1 227.148} C_DIS
LIN {X -0.088,Y -345.065,Z 1572.058,A 0.000,B 0.000,C 90.000,E1 226.377} C_DIS
LIN {X 0.094,Y -338.586,Z 1572.030,A 0.000,B 0.000,C 90.000,E1 221.310} C_DIS
LIN {X 0.094,Y -336.840,Z 1572.019,A 0.000,B 0.000,C 90.000,E1 219.358} C_DIS
LIN {X 0.014,Y -330.861,Z 1571.988,A 0.000,B 0.000,C 90.000,E1 213.865} C_DIS
LIN {X 0.149,Y -329.296,Z 1571.975,A 0.000,B 0.000,C 90.000,E1 211.465} C_DIS
LIN {X -0.154,Y -324.669,Z 1571.942,A 0.000,B 0.000,C 90.000,E1 205.540} C_DIS
LIN {X 0.174,Y -323.837,Z 1571.928,A 0.000,B 0.000,C 90.000,E1 203.078} C_DIS
LIN {X -0.017,Y -321.124,Z 1571.881,A 0.000,B 0.000,C 90.000,E1 194.662} C_DIS
LIN {X 0.138,Y -320.932,Z 1571.877,A 0.000,B 0.000,C 90.000,E1 193.828} C_DIS
LIN {X -0.076,Y -321.562,Z 1571.832,A 0.000,B 0.000,C 90.000,E1 185.796} C_DIS
LIN {X -0.143,Y -324.415,Z 1571.790,A 0.000,B 0.000,C 90.000,E1 178.165} C_DIS
LIN {X -0.141,Y -325.376,Z 1571.783,A 0.000,B 0.000,C 90.000,E1 176.963} C_DIS
LIN {X -0.100,Y -329.112,Z 1571.750,A 0.000,B 0.000,C 90.000,E1 170.971} C_DIS
LIN {X 0.061,Y -334.260,Z 1571.726,A 0.000,B 0.000,C 90.000,E1 166.589} C_DIS
LIN {X 0.067,Y -335.488,Z 1571.719,A 0.000,B 0.000,C 90.000,E1 165.408} C_DIS
LIN {X 0.143,Y -340.932,Z 1571.695,A 0.000,B 0.000,C 90.000,E1 161.094} C_DIS
LIN {X -0.172,Y -342.138,Z 1571.691,A 0.000,B 0.000,C 90.000,E1 160.369} C_DIS
LIN {X -0.058,Y -347.939,Z 1571.667,A 0.000,B 0.000,C 90.000,E1 156.102} C_DIS
LIN {X -0.081,Y -354.259,Z 1571.648,A 0.000,B 0.000,C 90.000,E1 152.666} C_DIS
LIN {X -0.222,Y -361.406,Z 1571.625,A 0.000,B 0.000,C 90.000,E1 148.535} C_DIS
LIN {X 0.065,Y -368.758,Z 1571.606,A 0.000,B 0.000,C 90.000,E1 145.135} C_DIS
LIN {X 0.065,Y -377.029,Z 1571.584,A 0.000,B 0.000,C 90.000,E1 141.090} C_DIS
LIN {X -0.061,Y -383.435,Z 1571.570,A 0.000,B 0.000,C 90.000,E1 138.566} C_DIS
LIN {X -0.015,Y -385.037,Z 1571.566,A 0.000,B 0.000,C 90.000,E1 137.838} C_DIS
LIN {X -0.004,Y -394.325,Z 1571.544,A 0.000,B 0.000,C 90.000,E1 133.905} C_DIS
LIN {X 0.107,Y -399.276,Z 1571.534,A 0.000,B 0.000,C 90.000,E1 132.123} C_DIS
LIN {X 0.210,Y -400.192,Z 1571.532,A 0.000,B 0.000,C 90.000,E1 131.757} C_DIS
LIN {X -0.113,Y -409.687,Z 1571.511,A 0.000,B 0.000,C 90.000,E1 127.971} C_DIS
LIN {X 0.046,Y -415.746,Z 1571.499,A 0.000,B 0.000,C 90.000,E1 125.884} C_DIS
LIN {X 0.153,Y -425.188,Z 1571.479,A 0.000,B 0.000,C 90.000,E1 122.133} C_DIS
LIN {X 0.087,Y -430.186,Z 1571.469,A 0.000,B 0.000,C 90.000,E1 120.463} C_DIS
LIN {X 0.086,Y -431.107,Z 1571.468,A 0.000,B 0.000,C 90.000,E1 120.129} C_DIS
LIN {X 0.032,Y -440.207,Z 1571.447,A 0.000,B 0.000,C 90.000,E1 116.488} C_DIS
LIN {X 0.039,Y -444.962,Z 1571.438,A 0.000,B 0.000,C 90.000,E1 114.847} C_DIS
LIN {X -0.108,Y -454.089,Z 1571.417,A 0.000,B 0.000,C 90.000,E1 110.972} C_DIS
LIN {X 0.005,Y -456.742,Z 1571.411,A 0.000,B 0.000,C 90.000,E1 109.993} C_DIS
LIN {X -0.096,Y -457.517,Z 1571.409,A 0.000,B 0.000,C 90.000,E1 109.685} C_DIS
LIN {X -0.146,Y -460.729,Z 1571.400,A 0.000,B 0.000,C 90.000,E1 108.000} C_DIS
LIN {X -0.208,Y -548.782,Z 1571.400,A 0.000,B 0.000,C 90.000,E1 108.000} C_DIS
LIN {X -0.243,Y -548.887,Z 1571.400,A 0.000,B 0.000,C 90.000,E1 108.000} C_DIS
LIN {X -0.083,Y -550.507,Z 1571.399,A 0.000,B 0.000,C 90.000,E1 107.764} C_DIS
LIN {X 0.173,Y -551.467,Z 1571.397,A 0.000,B 0.000,C 90.000,E1 107.457} C_DIS
LIN {X 0.008,Y -552.715,Z 1571.394,A 0.000,B 0.000,C 90.000,E1 106.913} C_DIS
LIN {X -0.039,Y -554.075,Z 1571.389,A 0.000,B 0.000,C 90.000,E1 106.079} C_DIS
LIN {X 0.052,Y -555.213,Z 1571.383,A 0.000,B 0.000,C 90.000,E1 104.954} C_DIS
LIN {X 0.030,Y -555.874,Z 1571.379,A 0.000,B 0.000,C 90.000,E1 104.120} C_DIS
LIN {X 0.149,Y -556.657,Z 1571.371,A 0.000,B 0.000,C 90.000,E1 102.715} C_DIS
LIN {X -0.115,Y -557.363,Z 1571.361,A 0.000,B 0.000,C 90.000,E1 101.074} C_DIS
LIN {X -0.108,Y -557.749,Z 1571.355,A 0.000,B 0.000,C 90.000,E1 99.962} C_DIS
LIN {X 0.080,Y -558.283,Z 1571.346,A 0.000,B 0.000,C 90.000,E1 98.276} C_DIS
LIN {X -0.143,Y -558.557,Z 1571.341,A 0.000,B 0.000,C 90.000,E1 97.466} C_DIS
LIN {X -0.093,Y -558.935,Z 1571.332,A 0.000,B 0.000,C 90.000,E1 95.796} C_DIS
LIN {X 0.045,Y -559.181,Z 1571.321,A 0.000,B 0.000,C 90.000,E1 93.841} C_DIS
LIN {X 0.036,Y -559.578,Z 1571.312,A 0.000,B 0.000,C 90.000,E1 92.178} C_DIS
LIN {X -0.053,Y -559.900,Z 1571.304,A 0.000,B 0.000,C 90.000,E1 90.802} C_DIS
LIN {X -0.057,Y -560.281,Z 1571.295,A 0.000,B 0.000,C 90.000,E1 89.141} C_DIS
LIN {X 0.143,Y -560.933,Z 1571.283,A 0.000,B 0.000,C 90.000,E1 86.906} C_DIS
LIN {X 0.196,Y -561.560,Z 1571.274,A 0.000,B 0.000,C 90.000,E1 85.241} C_DIS
LIN {X -0.098,Y -562.454,Z 1571.263,A 0.000,B 0.000,C 90.000,E1 83.337} C_DIS
LIN {X -0.206,Y -563.731,Z 1571.251,A 0.000,B 0.000,C 90.000,E1 81.141} C_DIS
LIN {X -0.099,Y -565.222,Z 1571.239,A 0.000,B 0.000,C 90.000,E1 78.926} C_DIS
LIN {X 0.198,Y -566.248,Z 1571.231,A 0.000,B 0.000,C 90.000,E1 77.521} C_DIS
LIN {X 0.129,Y -567.332,Z 1571.222,A 0.000,B 0.000,C 90.000,E1 75.880} C_DIS
LIN {X 0.031,Y -568.088,Z 1571.214,A 0.000,B 0.000,C 90.000,E1 74.519} C_DIS
LIN {X 0.103,Y -568.735,Z 1571.206,A 0.000,B 0.000,C 90.000,E1 73.142} C_DIS
LIN {X 0.023,Y -569.011,Z 1571.200,A 0.000,B 0.000,C 90.000,E1 72.054} C_DIS
LIN {X 0.105,Y -569.160,Z 1571.193,A 0.000,B 0.000,C 90.000,E1 70.678} C_DIS
LIN {X -0.169,Y -568.851,Z 1571.185,A 0.000,B 0.000,C 90.000,E1 69.337} C_DIS
LIN {X -0.011,Y -568.582,Z 1571.182,A 0.000,B 0.000,C 90.000,E1 68.773} C_DIS
LIN {X -0.060,Y -568.080,Z 1571.179,A 0.000,B 0.000,C 90.000,E1 68.230} C_DIS
LIN {X -0.245,Y -567.712,Z 1571.178,A 0.000,B 0.000,C 90.000,E1 67.975} C_DIS
LIN {X 0.097,Y -567.159,Z 1571.176,A 0.000,B 0.000,C 90.000,E1 67.667} C_DIS
LIN {X -0.087,Y -566.137,Z 1571.175,A 0.000,B 0.000,C 90.000,E1 67.411} C_DIS
LIN {X -0.148,Y -565.672,Z 1571.174,A 0.000,B 0.000,C 90.000,E1 67.358} C_DIS
LIN {X 0.092,Y -565.212,Z 1571.174,A 0.000,B 0.000,C 90.000,E1 67.305} C_DIS
LIN {X 0.029,Y -465.984,Z 1571.174,A 0.000,B 0.000,C 90.000,E1 67.305} C_DIS
LIN {X 0.207,Y -465.742,Z 1571.173,A 0.000,B 0.000,C 90.000,E1 67.102} C_DIS
LIN {X -0.048,Y -462.927,Z 1571.166,A 0.000,B 0.000,C 90.000,E1 65.869} C_DIS
LIN {X 0.107,Y -455.701,Z 1571.145,A 0.000,B 0.000,C 90.000,E1 62.025} C_DIS
LIN {X -0.004,Y -455.044,Z 1571.143,A 0.000,B 0.000,C 90.000,E1 61.719} C_DIS
LIN {X -0.177,Y -446.406,Z 1571.121,A 0.000,B 0.000,C 90.000,E1 57.867} C_DIS
LIN {X -0.047,Y -444.036,Z 1571.114,A 0.000,B 0.000,C 90.000,E1 56.548} C_DIS
LIN {X -0.002,Y -434.227,Z 1571.090,A 0.000,B 0.000,C 90.000,E1 52.271} C_DIS
LIN {X -0.159,Y -431.741,Z 1571.083,A 0.000,B 0.000,C 90.000,E1 50.964} C_DIS
LIN {X 0.021,Y -430.148,Z 1571.079,A 0.000,B 0.000,C 90.000,E1 50.275} C_DIS
LIN {X 0.155,Y -420.587,Z 1571.055,A 0.000,B 0.000,C 90.000,E1 45.891} C_DIS
LIN {X -0.169,Y -418.773,Z 1571.049,A 0.000,B 0.000,C 90.000,E1 44.919} C_DIS
LIN {X 0.092,Y -409.848,Z 1571.027,A 0.000,B 0.000,C 90.000,E1 40.782} C_DIS
LIN {X -0.046,Y -405.624,Z 1571.013,A 0.000,B 0.000,C 90.000,E1 38.382} C_DIS
LIN {X 0.017,Y -396.781,Z 1570.988,A 0.000,B 0.000,C 90.000,E1 33.833} C_DIS
LIN {X -0.008,Y -393.580,Z 1570.976,A 0.000,B 0.000,C 90.000,E1 31.720} C_DIS
LIN {X -0.100,Y -386.208,Z 1570.953,A 0.000,B 0.000,C 90.000,E1 27.462} C_DIS
LIN {X -0.122,Y -383.000,Z 1570.939,A 0.000,B 0.000,C 90.000,E1 24.951} C_DIS
LIN {X -0.019,Y -380.147,Z 1570.929,A 0.000,B 0.000,C 90.000,E1 23.131} C_DIS
LIN {X -0.146,Y -374.086,Z 1570.900,A 0.000,B 0.000,C 90.000,E1 18.055} C_DIS
LIN {X 0.161,Y -373.384,Z 1570.896,A 0.000,B 0.000,C 90.000,E1 17.275} C_DIS
LIN {X 0.176,Y -367.880,Z 1570.868,A 0.000,B 0.000,C 90.000,E1 12.119} C_DIS
LIN {X 0.120,Y -366.486,Z 1570.855,A 0.000,B 0.000,C 90.000,E1 9.905} C_DIS
LIN {X 0.056,Y -361.788,Z 1570.822,A 0.000,B 0.000,C 90.000,E1 3.955} C_DIS
LIN {X -0.059,Y -360.902,Z 1570.801,A 0.000,B 0.000,C 90.000,E1 0.229} C_DIS
LIN {X -0.053,Y -359.426,Z 1570.770,A 0.000,B 0.000,C 90.000,E1 354.546} C_DIS
LIN {X 0.070,Y -358.890,Z 1570.759,A 0.000,B 0.000,C 90.000,E1 352.648} C_DIS
LIN {X -0.020,Y -359.563,Z 1570.726,A 0.000,B 0.000,C 90.000,E1 346.645} C_DIS
LIN {X 0.001,Y -361.801,Z 1570.684,A 0.000,B 0.000,C 90.000,E1 339.135} C_DIS
LIN {X -0.154,Y -362.053,Z 1570.680,A 0.000,B 0.000,C 90.000,E1 338.411} C_DIS
LIN {X 0.189,Y -365.980,Z 1570.643,A 0.000,B 0.000,C 90.000,E1 331.641} C_DIS
LIN {X 0.029,Y -366.387,Z 1570.639,A 0.000,B 0.000,C 90.000,E1 330.923} C_DIS
LIN {X -0.031,Y -371.355,Z 1570.604,A 0.000,B 0.000,C 90.000,E1 324.642} C_DIS
LIN {X -0.043,Y -371.766,Z 1570.602,A 0.000,B 0.000,C 90.000,E1 324.276} C_DIS
LIN {X 0.013,Y -377.358,Z 1570.567,A 0.000,B 0.000,C 90.000,E1 318.038} C_DIS
LIN {X 0.012,Y -378.235,Z 1570.563,A 0.000,B 0.000,C 90.000,E1 317.310} C_DIS
LIN {X 0.002,Y -383.940,Z 1570.531,A 0.000,B 0.000,C 90.000,E1 311.515} C_DIS
LIN {X 0.088,Y -384.893,Z 1570.527,A 0.000,B 0.000,C 90.000,E1 310.782} C_DIS
LIN {X 0.262,Y -390.610,Z 1570.495,A 0.000,B 0.000,C 90.000,E1 305.025} C_DIS
LIN {X 0.106,Y -391.104,Z 1570.493,A 0.000,B 0.000,C 90.000,E1 304.692} C_DIS
LIN {X 0.022,Y -391.648,Z 1570.489,A 0.000,B 0.000,C 90.000,E1 303.992} C_DIS
LIN {X -0.080,Y -396.825,Z 1570.459,A 0.000,B 0.000,C 90.000,E1 298.693} C_DIS
LIN {X -0.210,Y -397.120,Z 1570.457,A 0.000,B 0.000,C 90.000,E1 298.359} C_DIS
LIN {X -0.055,Y -401.597,Z 1570.426,A 0.000,B 0.000,C 90.000,E1 292.717} C_DIS
LIN {X 0.222,Y -404.659,Z 1570.395,A 0.000,B 0.000,C 90.000,E1 287.094} C_DIS
LIN {X -0.079,Y -404.735,Z 1570.391,A 0.000,B 0.000,C 90.000,E1 286.441} C_DIS
LIN {X 0.214,Y -406.099,Z 1570.364,A 0.000,B 0.000,C 90.000,E1 281.535} C_DIS
LIN {X -0.176,Y -406.094,Z 1570.362,A 0.000,B 0.000,C 90.000,E1 281.243} C_DIS
LIN {X -0.097,Y -405.680,Z 1570.333,A 0.000,B 0.000,C 90.000,E1 276.024} C_DIS
LIN {X -0.165,Y -405.058,Z 1570.328,A 0.000,B 0.000,C 90.000,E1 274.992} C_DIS
LIN {X -0.060,Y -403.497,Z 1570.304,A 0.000,B 0.000,C 90.000,E1 270.802} C_DIS
LIN {X -0.092,Y -403.288,Z 1570.302,A 0.000,B 0.000,C 90.000,E1 270.458} C_DIS
LIN {X 0.091,Y -398.931,Z 1570.271,A 0.000,B 0.000,C 90.000,E1 264.837} C_DIS
LIN {X -0.040,Y -393.108,Z 1570.242,A 0.000,B 0.000,C 90.000,E1 259.567} C_DIS
LIN {X -0.079,Y -392.835,Z 1570.240,A 0.000,B 0.000,C 90.000,E1 259.218} C_DIS
LIN {X 0.034,Y -385.993,Z 1570.212,A 0.000,B 0.000,C 90.000,E1 254.212} C_DIS
LIN {X -0.026,Y -385.267,Z 1570.208,A 0.000,B 0.000,C 90.000,E1 253.504} C_DIS
LIN {X -0.004,Y -384.768,Z 1570.206,A 0.000,B 0.000,C 90.000,E1 253.142} C_DIS
LIN {X 0.221,Y -377.973,Z 1570.182,A 0.000,B 0.000,C 90.000,E1 248.773} C_DIS
LIN {X -0.044,Y -376.233,Z 1570.174,A 0.000,B 0.000,C 90.000,E1 247.358} C_DIS
LIN {X 0.057,Y -374.944,Z 1570.170,A 0.000,B 0.000,C 90.000,E1 246.613} C_DIS
LIN {X -0.208,Y -368.417,Z 1570.148,A 0.000,B 0.000,C 90.000,E1 242.615} C_DIS
LIN {X 0.097,Y -366.047,Z 1570.137,A 0.000,B 0.000,C 90.000,E1 240.717} C_DIS
LIN {X 0.004,Y -359.196,Z 1570.115,A 0.000,B 0.000,C 90.000,E1 236.628} C_DIS
LIN {X 0.021,Y -355.842,Z 1570.100,A 0.000,B 0.000,C 90.000,E1 233.989} C_DIS
LIN {X -0.173,Y -348.793,Z 1570.075,A 0.000,B 0.000,C 90.000,E1 229.461} C_DIS
LIN {X -0.097,Y -346.185,Z 1570.062,A 0.000,B 0.000,C 90.000,E1 227.148} C_DIS
LIN {X -0.088,Y -345.065,Z 1570.058,A 0.000,B 0.000,C 90.000,E1 226.377} C_DIS
LIN {X 0.094,Y -338.586,Z 1570.030,A 0.000,B 0.000,C 90.000,E1 221.310} C_DIS
LIN {X 0.094,Y -336.840,Z 1570.019,A 0.000,B 0.000,C 90.000,E1 219.358} C_DIS
LIN {X 0.014,Y -330.861,Z 1569.988,A 0.000,B 0.000,C 90.000,E1 213.865} C_DIS
LIN {X 0.149,Y -329.296,Z 1569.975,A 0.000,B 0.000,C 90.000,E1 211.465} C_DIS
LIN {X -0.154,Y -324.669,Z 1569.942,A 0.000,B 0.000,C 90.000,E1 205.540} C_DIS
LIN {X 0.174,Y -323.837,Z 1569.928,A 0.000,B 0.000,C 90.000,E1 203.078} C_DIS
LIN {X -0.017,Y -321.124,Z 1569.881,A 0.000,B 0.000,C 90.000,E1 194.662} C_DIS
LIN {X 0.138,Y -320.932,Z 1569.877,A 0.000,B 0.000,C 90.000,E1 193.828} C_DIS
LIN {X -0.076,Y -321.562,Z 1569.832,A 0.000,B 0.000,C 90.000,E1 185.796} C_DIS
LIN {X -0.143,Y -324.415,Z 1569.790,A 0.000,B 0.000,C 90.000,E1 178.165} C_DIS
LIN {X -0.141,Y -325.376,Z 1569.783,A 0.000,B 0.000,C 90.000,E1 176.963} C_DIS
LIN {X -0.100,Y -329.112,Z 1569.750,A 0.000,B 0.000,C 90.000,E1 170.971} C_DIS
LIN {X 0.061,Y -334.260,Z 1569.726,A 0.000,B 0.000,C 90.000,E1 166.589} C_DIS
LIN {X 0.067,Y -335.488,Z 1569.719,A 0.000,B 0.000,C 90.000,E1 165.408} C_DIS
LIN {X 0.143,Y -340.932,Z 1569.695,A 0.000,B 0.000,C 90.000,E1 161.094} C_DIS
LIN {X -0.172,Y -342.138,Z 1569.691,A 0.000,B 0.000,C 90.000,E1 160.369} C_DIS
LIN {X -0.058,Y -347.939,Z 1569.667,A 0.000,B 0.000,C 90.000,E1 156.102} C_DIS
LIN {X -0.081,Y -354.259,Z 1569.648,A 0.000,B 0.000,C 90.000,E1 152.666} C_DIS
LIN {X -0.222,Y -361.406,Z 1569.625,A 0.000,B 0.000,C 90.000,E1 148.535} C_DIS
LIN {X 0.065,Y -368.758,Z 1569.606,A 0.000,B 0.000,C 90.000,E1 145.135} C_DIS
LIN {X 0.065,Y -377.029,Z 1569.584,A 0.000,B 0.000,C 90.000,E1 141.090} C_DIS
LIN {X -0.061,Y -383.435,Z 1569.570,A 0.000,B 0.000,C 90.000,E1 138.566} C_DIS
LIN {X -0.015,Y -385.037,Z 1569.566,A 0.000,B 0.000,C 90.000,E1 137.838} C_DIS
LIN {X -0.004,Y -394.325,Z 1569.544,A 0.000,B 0.000,C 90.000,E1 133.905} C_DIS
LIN {X 0.107,Y -399.276,Z 1569.534,A 0.000,B 0.000,C 90.000,E1 132.123} C_DIS
LIN {X 0.210,Y -400.192,Z 1569.532,A 0.000,B 0.000,C 90.000,E1 131.757} C_DIS
LIN {X -0.113,Y -409.687,Z 1569.511,A 0.000,B 0.000,C 90.000,E1 127.971} C_DIS
LIN {X 0.046,Y -415.746,Z 1569.499,A 0.000,B 0.000,C 90.000,E1 125.884} C_DIS
LIN {X 0.153,Y -425.188,Z 1569.479,A 0.000,B 0.000,C 90.000,E1 122.133} C_DIS
LIN {X 0.087,Y -430.186,Z 1569.469,A 0.000,B 0.000,C 90.000,E1 120.463} C_DIS
LIN {X 0.086,Y -431.107,Z 1569.468,A 0.000,B 0.000,C 90.000,E1 120.129} C_DIS
LIN {X 0.032,Y -440.207,Z 1569.447,A 0.000,B 0.000,C 90.000,E1 116.488} C_DIS
LIN {X 0.039,Y -444.962,Z 1569.438,A 0.000,B 0.000,C 90.000,E1 114.847} C_DIS
LIN {X -0.108,Y -454.089,Z 1569.417,A 0.000,B 0.000,C 90.000,E1 110.972} C_DIS
LIN {X 0.194,Y -456.675,Z 1569.411,A 0.000,B 0.000,C 90.000,E1 109.993} C_DIS
LIN {X 0.185,Y -548.695,Z 1569.411,A 0.000,B 0.000,C 90.000,E1 109.993} C_DIS
LIN {X 0.004,Y -549.111,Z 1569.411,A 0.000,B 0.000,C 90.000,E1 109.993} C_DIS
LIN {X 0.273,Y -550.336,Z 1569.410,A 0.000,B 0.000,C 90.000,E1 109.812} C_DIS
LIN {X -0.168,Y -551.432,Z 1569.409,A 0.000,B 0.000,C 90.000,E1 109.577} C_DIS
LIN {X -0.152,Y -552.777,Z 1569.406,A 0.000,B 0.000,C 90.000,E1 109.014} C_DIS
LIN {X 0.216,Y -553.743,Z 1569.402,A 0.000,B 0.000,C 90.000,E1 108.417} C_DIS
LIN {X 0.177,Y -554.791,Z 1569.398,A 0.000,B 0.000,C 90.000,E1 107.583} C_DIS
LIN {X 0.023,Y -556.073,Z 1569.390,A 0.000,B 0.000,C 90.000,E1 106.205} C_DIS
LIN {X 0.146,Y -556.756,Z 1569.384,A 0.000,B 0.000,C 90.000,E1 105.079} C_DIS
LIN {X -0.260,Y -557.273,Z 1569.378,A 0.000,B 0.000,C 90.000,E1 104.008} C_DIS
LIN {X 0.011,Y -557.707,Z 1569.370,A 0.000,B 0.000,C 90.000,E1 102.591} C_DIS
LIN {X -0.242,Y -558.135,Z 1569.361,A 0.000,B 0.000,C 90.000,E1 100.950} C_DIS
LIN {X -0.185,Y -558.392,Z 1569.353,A 0.000,B 0.000,C 90.000,E1 99.557} C_DIS
LIN {X 0.016,Y -558.846,Z 1569.344,A 0.000,B 0.000,C 90.000,E1 97.871} C_DIS
LIN {X -0.133,Y -559.072,Z 1569.338,A 0.000,B 0.000,C 90.000,E1 96.777} C_DIS
LIN {X -0.275,Y -559.331,Z 1569.331,A 0.000,B 0.000,C 90.000,E1 95.682} C_DIS
LIN {X 0.226,Y -559.577,Z 1569.324,A 0.000,B 0.000,C 90.000,E1 94.245} C_DIS
LIN {X -0.212,Y -559.995,Z 1569.313,A 0.000,B 0.000,C 90.000,E1 92.350} C_DIS
LIN {X -0.200,Y -560.404,Z 1569.304,A 0.000,B 0.000,C 90.000,E1 90.688} C_DIS
LIN {X 0.273,Y -560.749,Z 1569.296,A 0.000,B 0.000,C 90.000,E1 89.255} C_DIS
LIN {X 0.051,Y -561.450,Z 1569.282,A 0.000,B 0.000,C 90.000,E1 86.788} C_DIS
LIN {X 0.129,Y -562.102,Z 1569.273,A 0.000,B 0.000,C 90.000,E1 85.122} C_DIS
LIN {X 0.207,Y -562.843,Z 1569.264,A 0.000,B 0.000,C 90.000,E1 83.457} C_DIS
LIN {X 0.020,Y -563.930,Z 1569.253,A 0.000,B 0.000,C 90.000,E1 81.546} C_DIS
LIN {X 0.030,Y -565.382,Z 1569.241,A 0.000,B 0.000,C 90.000,E1 79.342} C_DIS
LIN {X -0.058,Y -566.645,Z 1569.232,A 0.000,B 0.000,C 90.000,E1 77.701} C_DIS
LIN {X -0.124,Y -567.776,Z 1569.223,A 0.000,B 0.000,C 90.000,E1 76.061} C_DIS
LIN {X 0.109,Y -568.838,Z 1569.213,A 0.000,B 0.000,C 90.000,E1 74.393} C_DIS
LIN {X 0.201,Y -569.694,Z 1569.206,A 0.000,B 0.000,C 90.000,E1 73.015} C_DIS
LIN {X 0.307,Y -570.287,Z 1569.198,A 0.000,B 0.000,C 90.000,E1 71.638} C_DIS
LIN {X 0.247,Y -570.658,Z 1569.192,A 0.000,B 0.000,C 90.000,E1 70.550} C_DIS
LIN {X 0.003,Y -570.936,Z 1569.185,A 0.000,B 0.000,C 90.000,E1 69.209} C_DIS
LIN {X 0.145,Y -570.976,Z 1569.178,A 0.000,B 0.000,C 90.000,E1 68.103} C_DIS
LIN {X -0.069,Y -570.794,Z 1569.174,A 0.000,B 0.000,C 90.000,E1 67.305} C_DIS
LIN {X 0.109,Y -570.553,Z 1569.171,A 0.000,B 0.000,C 90.000,E1 66.741} C_DIS
LIN {X -0.235,Y -570.052,Z 1569.168,A 0.000,B 0.000,C 90.000,E1 66.230} C_DIS
LIN {X -0.058,Y -569.148,Z 1569.165,A 0.000,B 0.000,C 90.000,E1 65.665} C_DIS
LIN {X -0.009,Y -568.074,Z 1569.163,A 0.000,B 0.000,C 90.000,E1 65.357} C_DIS
LIN {X 0.174,Y -567.651,Z 1569.163,A 0.000,B 0.000,C 90.000,E1 65.281} C_DIS
LIN {X 0.298,Y -567.049,Z 1569.163,A 0.000,B 0.000,C 90.000,E1 65.229} C_DIS
LIN {X 0.263,Y -566.875,Z 1569.163,A 0.000,B 0.000,C 90.000,E1 65.229} C_DIS
LIN {X 0.185,Y -461.615,Z 1569.163,A 0.000,B 0.000,C 90.000,E1 65.229} C_DIS
LIN {X 0.187,Y -455.514,Z 1569.144,A 0.000,B 0.000,C 90.000,E1 61.897} C_DIS
LIN {X 0.193,Y -445.567,Z 1569.119,A 0.000,B 0.000,C 90.000,E1 57.375} C_DIS
LIN {X 0.009,Y -443.784,Z 1569.114,A 0.000,B 0.000,C 90.000,E1 56.421} C_DIS
LIN {X 0.022,Y -434.645,Z 1569.092,A 0.000,B 0.000,C 90.000,E1 52.477} C_DIS
LIN {X 0.134,Y -431.520,Z 1569.082,A 0.000,B 0.000,C 90.000,E1 50.803} C_DIS
LIN {X 0.042,Y -421.634,Z 1569.058,A 0.000,B 0.000,C 90.000,E1 46.458} C_DIS
LIN {X 0.103,Y -418.530,Z 1569.049,A 0.000,B 0.000,C 90.000,E1 44.757} C_DIS
LIN {X -0.076,Y -408.975,Z 1569.024,A 0.000,B 0.000,C 90.000,E1 40.334} C_DIS
LIN {X 0.049,Y -406.044,Z 1569.015,A 0.000,B 0.000,C 90.000,E1 38.588} C_DIS
LIN {X 0.043,Y -398.968,Z 1568.995,A 0.000,B 0.000,C 90.000,E1 35.105} C_DIS
LIN {X 0.110,Y -393.944,Z 1568.978,A 0.000,B 0.000,C 90.000,E1 31.926} C_DIS
LIN {X -0.052,Y -390.619,Z 1568.968,A 0.000,B 0.000,C 90.000,E1 30.178} C_DIS
LIN {X -0.129,Y -383.677,Z 1568.942,A 0.000,B 0.000,C 90.000,E1 25.540} C_DIS
LIN {X 0.195,Y -382.846,Z 1568.938,A 0.000,B 0.000,C 90.000,E1 24.771} C_DIS
LIN {X 0.149,Y -376.142,Z 1568.912,A 0.000,B 0.000,C 90.000,E1 20.066} C_DIS
LIN {X 0.134,Y -373.664,Z 1568.897,A 0.000,B 0.000,C 90.000,E1 17.511} C_DIS
LIN {X 0.162,Y -368.060,Z 1568.869,A 0.000,B 0.000,C 90.000,E1 12.355} C_DIS
LIN {X -0.030,Y -366.372,Z 1568.854,A 0.000,B 0.000,C 90.000,E1 9.792} C_DIS
LIN {X -0.090,Y -361.727,Z 1568.821,A 0.000,B 0.000,C 90.000,E1 3.841} C_DIS
LIN {X 0.157,Y -360.845,Z 1568.801,A 0.000,B 0.000,C 90.000,E1 0.057} C_DIS
LIN {X -0.053,Y -359.426,Z 1568.770,A 0.000,B 0.000,C 90.000,E1 354.546} C_DIS
LIN {X 0.070,Y -358.890,Z 1568.759,A 0.000,B 0.000,C 90.000,E1 352.648} C_DIS
LIN {X -0.020,Y -359.563,Z 1568.726,A 0.000,B 0.000,C 90.000,E1 346.645} C_DIS
LIN {X 0.001,Y -361.801,Z 1568.684,A 0.000,B 0.000,C 90.000,E1 339.135} C_DIS
LIN {X -0.154,Y -362.053,Z 1568.680,A 0.000,B 0.000,C 90.000,E1 338.411} C_DIS
LIN {X 0.189,Y -365.980,Z 1568.643,A 0.000,B 0.000,C 90.000,E1 331.641} C_DIS
LIN {X 0.029,Y -366.387,Z 1568.639,A 0.000,B 0.000,C 90.000,E1 330.923} C_DIS
LIN {X -0.031,Y -371.355,Z 1568.604,A 0.000,B 0.000,C 90.000,E1 324.642} C_DIS
LIN {X -0.043,Y -371.766,Z 1568.602,A 0.000,B 0.000,C 90.000,E1 324.276} C_DIS
LIN {X 0.013,Y -377.358,Z 1568.567,A 0.000,B 0.000,C 90.000,E1 318.038} C_DIS
LIN {X 0.012,Y -378.235,Z 1568.563,A 0.000,B 0.000,C 90.000,E1 317.310} C_DIS
LIN {X 0.002,Y -383.940,Z 1568.531,A 0.000,B 0.000,C 90.000,E1 311.515} C_DIS
LIN {X 0.088,Y -384.893,Z 1568.527,A 0.000,B 0.000,C 90.000,E1 310.782} C_DIS
LIN {X 0.262,Y -390.610,Z 1568.495,A 0.000,B 0.000,C 90.000,E1 305.025} C_DIS
LIN {X 0.106,Y -391.104,Z 1568.493,A 0.000,B 0.000,C 90.000,E1 304.692} C_DIS
LIN {X 0.022,Y -391.648,Z 1568.489,A 0.000,B 0.000,C 90.000,E1 303.992} C_DIS
LIN {X -0.080,Y -396.825,Z 1568.459,A 0.000,B 0.000,C 90.000,E1 298.693} C_DIS
LIN {X -0.210,Y -397.120,Z 1568.457,A 0.000,B 0.000,C 90.000,E1 298.359} C_DIS
LIN {X -0.055,Y -401.597,Z 1568.426,A 0.000,B 0.000,C 90.000,E1 292.717} C_DIS
LIN {X 0.222,Y -404.659,Z 1568.395,A 0.000,B 0.000,C 90.000,E1 287.094} C_DIS
LIN {X -0.079,Y -404.735,Z 1568.391,A 0.000,B 0.000,C 90.000,E1 286.441} C_DIS
LIN {X 0.214,Y -406.099,Z 1568.364,A 0.000,B 0.000,C 90.000,E1 281.535} C_DIS
LIN {X -0.176,Y -406.094,Z 1568.362,A 0.000,B 0.000,C 90.000,E1 281.243} C_DIS
LIN {X -0.097,Y -405.680,Z 1568.333,A 0.000,B 0.000,C 90.000,E1 276.024} C_DIS
LIN {X -0.165,Y -405.058,Z 1568.328,A 0.000,B 0.000,C 90.000,E1 274.992} C_DIS
LIN {X -0.060,Y -403.497,Z 1568.304,A 0.000,B 0.000,C 90.000,E1 270.802} C_DIS
LIN {X -0.092,Y -403.288,Z 1568.302,A 0.000,B 0.000,C 90.000,E1 270.458} C_DIS
LIN {X 0.091,Y -398.931,Z 1568.271,A 0.000,B 0.000,C 90.000,E1 264.837} C_DIS
LIN {X -0.040,Y -393.108,Z 1568.242,A 0.000,B 0.000,C 90.000,E1 259.567} C_DIS
LIN {X -0.079,Y -392.835,Z 1568.240,A 0.000,B 0.000,C 90.000,E1 259.218} C_DIS
LIN {X 0.034,Y -385.993,Z 1568.212,A 0.000,B 0.000,C 90.000,E1 254.212} C_DIS
LIN {X -0.026,Y -385.267,Z 1568.208,A 0.000,B 0.000,C 90.000,E1 253.504} C_DIS
LIN {X -0.004,Y -384.768,Z 1568.206,A 0.000,B 0.000,C 90.000,E1 253.142} C_DIS
LIN {X 0.221,Y -377.973,Z 1568.182,A 0.000,B 0.000,C 90.000,E1 248.773} C_DIS
LIN {X -0.044,Y -376.233,Z 1568.174,A 0.000,B 0.000,C 90.000,E1 247.358} C_DIS
LIN {X 0.057,Y -374.944,Z 1568.170,A 0.000,B 0.000,C 90.000,E1 246.613} C_DIS
LIN {X -0.208,Y -368.417,Z 1568.148,A 0.000,B 0.000,C 90.000,E1 242.615} C_DIS
LIN {X 0.097,Y -366.047,Z 1568.137,A 0.000,B 0.000,C 90.000,E1 240.717} C_DIS
LIN {X 0.004,Y -359.196,Z 1568.115,A 0.000,B 0.000,C 90.000,E1 236.628} C_DIS
LIN {X 0.021,Y -355.842,Z 1568.100,A 0.000,B 0.000,C 90.000,E1 233.989} C_DIS
LIN {X -0.173,Y -348.793,Z 1568.075,A 0.000,B 0.000,C 90.000,E1 229.461} C_DIS
LIN {X -0.097,Y -346.185,Z 1568.062,A 0.000,B 0.000,C 90.000,E1 227.148} C_DIS
LIN {X -0.088,Y -345.065,Z 1568.058,A 0.000,B 0.000,C 90.000,E1 226.377} C_DIS
LIN {X 0.094,Y -338.586,Z 1568.030,A 0.000,B 0.000,C 90.000,E1 221.310} C_DIS
LIN {X 0.094,Y -336.840,Z 1568.019,A 0.000,B 0.000,C 90.000,E1 219.358} C_DIS
LIN {X 0.014,Y -330.861,Z 1567.988,A 0.000,B 0.000,C 90.000,E1 213.865} C_DIS
LIN {X 0.149,Y -329.296,Z 1567.975,A 0.000,B 0.000,C 90.000,E1 211.465} C_DIS
LIN {X -0.154,Y -324.669,Z 1567.942,A 0.000,B 0.000,C 90.000,E1 205.540} C_DIS
LIN {X 0.174,Y -323.837,Z 1567.928,A 0.000,B 0.000,C 90.000,E1 203.078} C_DIS
LIN {X -0.017,Y -321.124,Z 1567.881,A 0.000,B 0.000,C 90.000,E1 194.662} C_DIS
LIN {X 0.138,Y -320.932,Z 1567.877,A 0.000,B 0.000,C 90.000,E1 193.828} C_DIS
LIN {X -0.076,Y -321.562,Z 1567.832,A 0.000,B 0.000,C 90.000,E1 185.796} C_DIS
LIN {X -0.143,Y -324.415,Z 1567.790,A 0.000,B 0.000,C 90.000,E1 178.165} C_DIS
LIN {X -0.141,Y -325.376,Z 1567.783,A 0.000,B 0.000,C 90.000,E1 176.963} C_DIS
LIN {X -0.100,Y -329.112,Z 1567.750,A 0.000,B 0.000,C 90.000,E1 170.971} C_DIS
LIN {X 0.061,Y -334.260,Z 1567.726,A 0.000,B 0.000,C 90.000,E1 166.589} C_DIS
LIN {X 0.067,Y -335.488,Z 1567.719,A 0.000,B 0.000,C 90.000,E1 165.408} C_DIS
LIN {X 0.143,Y -340.932,Z 1567.695,A 0.000,B 0.000,C 90.000,E1 161.094} C_DIS
LIN {X -0.172,Y -342.138,Z 1567.691,A 0.000,B 0.000,C 90.000,E1 160.369} C_DIS
LIN {X -0.058,Y -347.939,Z 1567.667,A 0.000,B 0.000,C 90.000,E1 156.102} C_DIS
LIN {X -0.081,Y -354.259,Z 1567.648,A 0.000,B 0.000,C 90.000,E1 152.666} C_DIS
LIN {X -0.222,Y -361.406,Z 1567.625,A 0.000,B 0.000,C 90.000,E1 148.535} C_DIS
LIN {X 0.065,Y -368.758,Z 1567.606,A 0.000,B 0.000,C 90.000,E1 145.135} C_DIS
LIN {X 0.065,Y -377.029,Z 1567.584,A 0.000,B 0.000,C 90.000,E1 141.090} C_DIS
LIN {X -0.061,Y -383.435,Z 1567.570,A 0.000,B 0.000,C 90.000,E1 138.566} C_DIS
LIN {X -0.015,Y -385.037,Z 1567.566,A 0.000,B 0.000,C 90.000,E1 137.838} C_DIS
LIN {X -0.004,Y -394.325,Z 1567.544,A 0.000,B 0.000,C 90.000,E1 133.905} C_DIS
LIN {X 0.107,Y -399.276,Z 1567.534,A 0.000,B 0.000,C 90.000,E1 132.123} C_DIS
LIN {X 0.210,Y -400.192,Z 1567.532,A 0.000,B 0.000,C 90.000,E1 131.757} C_DIS
LIN {X -0.113,Y -409.687,Z 1567.511,A 0.000,B 0.000,C 90.000,E1 127.971} C_DIS
LIN {X 0.046,Y -415.746,Z 1567.499,A 0.000,B 0.000,C 90.000,E1 125.884} C_DIS
LIN {X 0.153,Y -425.188,Z 1567.479,A 0.000,B 0.000,C 90.000,E1 122.133} C_DIS
LIN {X 0.087,Y -430.186,Z 1567.469,A 0.000,B 0.000,C 90.000,E1 120.463} C_DIS
LIN {X 0.086,Y -431.107,Z 1567.468,A 0.000,B 0.000,C 90.000,E1 120.129} C_DIS
LIN {X 0.032,Y -440.207,Z 1567.447,A 0.000,B 0.000,C 90.000,E1 116.488} C_DIS
LIN {X 0.039,Y -444.962,Z 1567.438,A 0.000,B 0.000,C 90.000,E1 114.847} C_DIS
LIN {X -0.101,Y -451.690,Z 1567.422,A 0.000,B 0.000,C 90.000,E1 111.897} C_DIS
LIN {X -0.159,Y -548.655,Z 1567.422,A 0.000,B 0.000,C 90.000,E1 111.897} C_DIS
LIN {X 0.229,Y -550.120,Z 1567.421,A 0.000,B 0.000,C 90.000,E1 111.716} C_DIS
LIN {X 0.141,Y -550.792,Z 1567.420,A 0.000,B 0.000,C 90.000,E1 111.589} C_DIS
LIN {X -0.103,Y -551.758,Z 1567.418,A 0.000,B 0.000,C 90.000,E1 111.334} C_DIS
LIN {X 0.244,Y -553.121,Z 1567.415,A 0.000,B 0.000,C 90.000,E1 110.737} C_DIS
LIN {X 0.137,Y -554.787,Z 1567.409,A 0.000,B 0.000,C 90.000,E1 109.631} C_DIS
LIN {X -0.138,Y -555.866,Z 1567.403,A 0.000,B 0.000,C 90.000,E1 108.544} C_DIS
LIN {X 0.136,Y -556.633,Z 1567.397,A 0.000,B 0.000,C 90.000,E1 107.402} C_DIS
LIN {X 0.010,Y -557.388,Z 1567.389,A 0.000,B 0.000,C 90.000,E1 106.024} C_DIS
LIN {X -0.113,Y -557.827,Z 1567.381,A 0.000,B 0.000,C 90.000,E1 104.647} C_DIS
LIN {X -0.246,Y -558.000,Z 1567.377,A 0.000,B 0.000,C 90.000,E1 103.828} C_DIS
LIN {X 0.034,Y -558.221,Z 1567.369,A 0.000,B 0.000,C 90.000,E1 102.411} C_DIS
LIN {X -0.320,Y -558.538,Z 1567.360,A 0.000,B 0.000,C 90.000,E1 100.782} C_DIS
LIN {X 0.179,Y -559.075,Z 1567.347,A 0.000,B 0.000,C 90.000,E1 98.511} C_DIS
LIN {X 0.175,Y -559.434,Z 1567.340,A 0.000,B 0.000,C 90.000,E1 97.125} C_DIS
LIN {X -0.301,Y -559.723,Z 1567.330,A 0.000,B 0.000,C 90.000,E1 95.511} C_DIS
LIN {X 0.211,Y -560.048,Z 1567.323,A 0.000,B 0.000,C 90.000,E1 94.073} C_DIS
LIN {X 0.256,Y -560.442,Z 1567.314,A 0.000,B 0.000,C 90.000,E1 92.407} C_DIS
LIN {X 0.276,Y -560.842,Z 1567.304,A 0.000,B 0.000,C 90.000,E1 90.745} C_DIS
LIN {X 0.197,Y -561.224,Z 1567.297,A 0.000,B 0.000,C 90.000,E1 89.370} C_DIS
LIN {X -0.040,Y -561.889,Z 1567.283,A 0.000,B 0.000,C 90.000,E1 86.906} C_DIS
LIN {X 0.174,Y -562.669,Z 1567.272,A 0.000,B 0.000,C 90.000,E1 84.951} C_DIS
LIN {X 0.002,Y -563.718,Z 1567.260,A 0.000,B 0.000,C 90.000,E1 82.761} C_DIS
LIN {X 0.010,Y -564.984,Z 1567.248,A 0.000,B 0.000,C 90.000,E1 80.557} C_DIS
LIN {X 0.159,Y -566.650,Z 1567.235,A 0.000,B 0.000,C 90.000,E1 78.342} C_DIS
LIN {X 0.280,Y -568.045,Z 1567.225,A 0.000,B 0.000,C 90.000,E1 76.408} C_DIS
LIN {X 0.001,Y -569.273,Z 1567.214,A 0.000,B 0.000,C 90.000,E1 74.519} C_DIS
LIN {X -0.279,Y -570.306,Z 1567.205,A 0.000,B 0.000,C 90.000,E1 72.906} C_DIS
LIN {X -0.013,Y -571.342,Z 1567.194,A 0.000,B 0.000,C 90.000,E1 70.967} C_DIS
LIN {X -0.259,Y -572.213,Z 1567.184,A 0.000,B 0.000,C 90.000,E1 69.082} C_DIS
LIN {X 0.264,Y -572.666,Z 1567.176,A 0.000,B 0.000,C 90.000,E1 67.667} C_DIS
LIN {X -0.100,Y -572.842,Z 1567.170,A 0.000,B 0.000,C 90.000,E1 66.613} C_DIS
LIN {X -0.233,Y -572.728,Z 1567.164,A 0.000,B 0.000,C 90.000,E1 65.537} C_DIS
LIN {X -0.037,Y -572.516,Z 1567.161,A 0.000,B 0.000,C 90.000,E1 64.973} C_DIS
LIN {X 0.155,Y -571.891,Z 1567.158,A 0.000,B 0.000,C 90.000,E1 64.409} C_DIS
LIN {X -0.009,Y -571.486,Z 1567.156,A 0.000,B 0.000,C 90.000,E1 64.152} C_DIS
LIN {X -0.173,Y -570.932,Z 1567.155,A 0.000,B 0.000,C 90.000,E1 63.896} C_DIS
LIN {X -0.123,Y -569.919,Z 1567.153,A 0.000,B 0.000,C 90.000,E1 63.589} C_DIS
LIN {X 0.057,Y -569.163,Z 1567.153,A 0.000,B 0.000,C 90.000,E1 63.461} C_DIS
LIN {X -0.071,Y -568.439,Z 1567.152,A 0.000,B 0.000,C 90.000,E1 63.435} C_DIS
LIN {X -0.087,Y -458.053,Z 1567.152,A 0.000,B 0.000,C 90.000,E1 63.435} C_DIS
LIN {X 0.222,Y -455.725,Z 1567.145,A 0.000,B 0.000,C 90.000,E1 62.025} C_DIS
LIN {X 0.111,Y -455.081,Z 1567.143,A 0.000,B 0.000,C 90.000,E1 61.719} C_DIS
LIN {X -0.061,Y -446.435,Z 1567.121,A 0.000,B 0.000,C 90.000,E1 57.867} C_DIS
LIN {X 0.068,Y -444.060,Z 1567.114,A 0.000,B 0.000,C 90.000,E1 56.548} C_DIS
LIN {X 0.112,Y -434.258,Z 1567.091,A 0.000,B 0.000,C 90.000,E1 52.271} C_DIS
LIN {X -0.045,Y -431.768,Z 1567.083,A 0.000,B 0.000,C 90.000,E1 50.964} C_DIS
LIN {X 0.135,Y -430.186,Z 1567.079,A 0.000,B 0.000,C 90.000,E1 50.275} C_DIS
LIN {X 0.267,Y -420.615,Z 1567.055,A 0.000,B 0.000,C 90.000,E1 45.891} C_DIS
LIN {X -0.056,Y -418.799,Z 1567.050,A 0.000,B 0.000,C 90.000,E1 44.919} C_DIS
LIN {X 0.020,Y -411.903,Z 1567.032,A 0.000,B 0.000,C 90.000,E1 41.838} C_DIS
LIN {X 0.066,Y -405.660,Z 1567.013,A 0.000,B 0.000,C 90.000,E1 38.382} C_DIS
LIN {X 0.031,Y -397.388,Z 1566.990,A 0.000,B 0.000,C 90.000,E1 34.199} C_DIS
LIN {X -0.105,Y -393.613,Z 1566.976,A 0.000,B 0.000,C 90.000,E1 31.750} C_DIS
LIN {X 0.009,Y -386.232,Z 1566.953,A 0.000,B 0.000,C 90.000,E1 27.462} C_DIS
LIN {X -0.013,Y -383.019,Z 1566.939,A 0.000,B 0.000,C 90.000,E1 24.951} C_DIS
LIN {X -0.207,Y -381.300,Z 1566.933,A 0.000,B 0.000,C 90.000,E1 23.898} C_DIS
LIN {X 0.026,Y -375.135,Z 1566.906,A 0.000,B 0.000,C 90.000,E1 19.141} C_DIS
LIN {X -0.087,Y -373.407,Z 1566.896,A 0.000,B 0.000,C 90.000,E1 17.330} C_DIS
LIN {X -0.076,Y -367.893,Z 1566.868,A 0.000,B 0.000,C 90.000,E1 12.175} C_DIS
LIN {X -0.133,Y -366.495,Z 1566.855,A 0.000,B 0.000,C 90.000,E1 9.962} C_DIS
LIN {X 0.164,Y -361.796,Z 1566.822,A 0.000,B 0.000,C 90.000,E1 3.955} C_DIS
LIN {X 0.049,Y -360.903,Z 1566.801,A 0.000,B 0.000,C 90.000,E1 0.229} C_DIS
LIN {X -0.053,Y -359.426,Z 1566.770,A 0.000,B 0.000,C 90.000,E1 354.546} C_DIS
LIN {X 0.070,Y -358.890,Z 1566.759,A 0.000,B 0.000,C 90.000,E1 352.648} C_DIS
LIN {X -0.020,Y -359.563,Z 1566.726,A 0.000,B 0.000,C 90.000,E1 346.645} C_DIS
LIN {X 0.001,Y -361.801,Z 1566.684,A 0.000,B 0.000,C 90.000,E1 339.135} C_DIS
LIN {X -0.154,Y -362.053,Z 1566.680,A 0.000,B 0.000,C 90.000,E1 338.411} C_DIS
LIN {X 0.189,Y -365.980,Z 1566.643,A 0.000,B 0.000,C 90.000,E1 331.641} C_DIS
LIN {X 0.029,Y -366.387,Z 1566.639,A 0.000,B 0.000,C 90.000,E1 330.923} C_DIS
LIN {X -0.031,Y -371.355,Z 1566.604,A 0.000,B 0.000,C 90.000,E1 324.642} C_DIS
LIN {X -0.043,Y -371.766,Z 1566.602,A 0.000,B 0.000,C 90.000,E1 324.276} C_DIS
LIN {X 0.013,Y -377.358,Z 1566.567,A 0.000,B 0.000,C 90.000,E1 318.038} C_DIS
LIN {X 0.012,Y -378.235,Z 1566.563,A 0.000,B 0.000,C 90.000,E1 317.310} C_DIS
LIN {X 0.002,Y -383.940,Z 1566.531,A 0.000,B 0.000,C 90.000,E1 311.515} C_DIS
LIN {X 0.088,Y -384.893,Z 1566.527,A 0.000,B 0.000,C 90.000,E1 310.782} C_DIS
LIN {X 0.262,Y -390.610,Z 1566.495,A 0.000,B 0.000,C 90.000,E1 305.025} C_DIS
LIN {X 0.106,Y -391.104,Z 1566.493,A 0.000,B 0.000,C 90.000,E1 304.692} C_DIS
LIN {X 0.022,Y -391.648,Z 1566.489,A 0.000,B 0.000,C 90.000,E1 303.992} C_DIS
LIN {X -0.080,Y -396.825,Z 1566.459,A 0.000,B 0.000,C 90.000,E1 298.693} C_DIS
LIN {X -0.210,Y -397.120,Z 1566.457,A 0.000,B 0.000,C 90.000,E1 298.359} C_DIS
LIN {X -0.055,Y -401.597,Z 1566.426,A 0.000,B 0.000,C 90.000,E1 292.717} C_DIS
LIN {X 0.222,Y -404.659,Z 1566.395,A 0.000,B 0.000,C 90.000,E1 287.094} C_DIS
LIN {X -0.079,Y -404.735,Z 1566.391,A 0.000,B 0.000,C 90.000,E1 286.441} C_DIS
LIN {X 0.214,Y -406.099,Z 1566.364,A 0.000,B 0.000,C 90.000,E1 281.535} C_DIS
LIN {X -0.176,Y -406.094,Z 1566.362,A 0.000,B 0.000,C 90.000,E1 281.243} C_DIS
LIN {X -0.097,Y -405.680,Z 1566.333,A 0.000,B 0.000,C 90.000,E1 276.024} C_DIS
LIN {X -0.165,Y -405.058,Z 1566.328,A 0.000,B 0.000,C 90.000,E1 274.992} C_DIS
LIN {X -0.060,Y -403.497,Z 1566.304,A 0.000,B 0.000,C 90.000,E1 270.802} C_DIS
LIN {X -0.092,Y -403.288,Z 1566.302,A 0.000,B 0.000,C 90.000,E1 270.458} C_DIS
LIN {X 0.091,Y -398.931,Z 1566.271,A 0.000,B 0.000,C 90.000,E1 264.837} C_DIS
LIN {X -0.040,Y -393.108,Z 1566.242,A 0.000,B 0.000,C 90.000,E1 259.567} C_DIS
LIN {X -0.079,Y -392.835,Z 1566.240,A 0.000,B 0.000,C 90.000,E1 259.218} C_DIS
LIN {X 0.034,Y -385.993,Z 1566.212,A 0.000,B 0.000,C 90.000,E1 254.212} C_DIS
LIN {X -0.026,Y -385.267,Z 1566.208,A 0.000,B 0.000,C 90.000,E1 253.504} C_DIS
LIN {X -0.004,Y -384.768,Z 1566.206,A 0.000,B 0.000,C 90.000,E1 253.142} C_DIS
LIN {X 0.221,Y -377.973,Z 1566.182,A 0.000,B 0.000,C 90.000,E1 248.773} C_DIS
LIN {X -0.044,Y -376.233,Z 1566.174,A 0.000,B 0.000,C 90.000,E1 247.358} C_DIS
LIN {X 0.057,Y -374.944,Z 1566.170,A 0.000,B 0.000,C 90.000,E1 246.613} C_DIS
LIN {X -0.208,Y -368.417,Z 1566.148,A 0.000,B 0.000,C 90.000,E1 242.615} C_DIS
LIN {X 0.097,Y -366.047,Z 1566.137,A 0.000,B 0.000,C 90.000,E1 240.717} C_DIS
LIN {X 0.004,Y -359.196,Z 1566.115,A 0.000,B 0.000,C 90.000,E1 236.628} C_DIS
LIN {X 0.021,Y -355.842,Z 1566.100,A 0.000,B 0.000,C 90.000,E1 233.989} C_DIS
LIN {X -0.173,Y -348.793,Z 1566.075,A 0.000,B 0.000,C 90.000,E1 229.461} C_DIS
LIN {X -0.097,Y -346.185,Z 1566.062,A 0.000,B 0.000,C 90.000,E1 227.148} C_DIS
LIN {X -0.088,Y -345.065,Z 1566.058,A 0.000,B 0.000,C 90.000,E1 226.377} C_DIS
LIN {X 0.094,Y -338.586,Z 1566.030,A 0.000,B 0.000,C 90.000,E1 221.310} C_DIS
LIN {X 0.094,Y -336.840,Z 1566.019,A 0.000,B 0.000,C 90.000,E1 219.358} C_DIS
LIN {X 0.014,Y -330.861,Z 1565.988,A 0.000,B 0.000,C 90.000,E1 213.865} C_DIS
LIN {X 0.149,Y -329.296,Z 1565.975,A 0.000,B 0.000,C 90.000,E1 211.465} C_DIS
LIN {X -0.154,Y -324.669,Z 1565.942,A 0.000,B 0.000,C 90.000,E1 205.540} C_DIS
LIN {X 0.174,Y -323.837,Z 1565.928,A 0.000,B 0.000,C 90.000,E1 203.078} C_DIS
LIN {X -0.017,Y -321.124,Z 1565.881,A 0.000,B 0.000,C 90.000,E1 194.662} C_DIS
LIN {X 0.138,Y -320.932,Z 1565.877,A 0.000,B 0.000,C 90.000,E1 193.828} C_DIS
LIN {X -0.076,Y -321.562,Z 1565.832,A 0.000,B 0.000,C 90.000,E1 185.796} C_DIS
LIN {X -0.143,Y -324.415,Z 1565.790,A 0.000,B 0.000,C 90.000,E1 178.165} C_DIS
LIN {X -0.141,Y -325.376,Z 1565.783,A 0.000,B 0.000,C 90.000,E1 176.963} C_DIS
LIN {X -0.100,Y -329.112,Z 1565.750,A 0.000,B 0.000,C 90.000,E1 170.971} C_DIS
LIN {X 0.061,Y -334.260,Z 1565.726,A 0.000,B 0.000,C 90.000,E1 166.589} C_DIS
LIN {X 0.067,Y -335.488,Z 1565.719,A 0.000,B 0.000,C 90.000,E1 165.408} C_DIS
LIN {X 0.143,Y -340.932,Z 1565.695,A 0.000,B 0.000,C 90.000,E1 161.094} C_DIS
LIN {X -0.172,Y -342.138,Z 1565.691,A 0.000,B 0.000,C 90.000,E1 160.369} C_DIS
LIN {X -0.058,Y -347.939,Z 1565.667,A 0.000,B 0.000,C 90.000,E1 156.102} C_DIS
LIN {X -0.081,Y -354.259,Z 1565.648,A 0.000,B 0.000,C 90.000,E1 152.666} C_DIS
LIN {X -0.222,Y -361.406,Z 1565.625,A 0.000,B 0.000,C 90.000,E1 148.535} C_DIS
LIN {X 0.065,Y -368.758,Z 1565.606,A 0.000,B 0.000,C 90.000,E1 145.135} C_DIS
LIN {X 0.065,Y -377.029,Z 1565.584,A 0.000,B 0.000,C 90.000,E1 141.090} C_DIS
LIN {X -0.061,Y -383.435,Z 1565.570,A 0.000,B 0.000,C 90.000,E1 138.566} C_DIS
LIN {X -0.015,Y -385.037,Z 1565.566,A 0.000,B 0.000,C 90.000,E1 137.838} C_DIS
LIN {X -0.004,Y -394.325,Z 1565.544,A 0.000,B 0.000,C 90.000,E1 133.905} C_DIS
LIN {X 0.107,Y -399.276,Z 1565.534,A 0.000,B 0.000,C 90.000,E1 132.123} C_DIS
LIN {X 0.210,Y -400.192,Z 1565.532,A 0.000,B 0.000,C 90.000,E1 131.757} C_DIS
LIN {X -0.113,Y -409.687,Z 1565.511,A 0.000,B 0.000,C 90.000,E1 127.971} C_DIS
LIN {X 0.046,Y -415.746,Z 1565.499,A 0.000,B 0.000,C 90.000,E1 125.884} C_DIS
LIN {X 0.153,Y -425.188,Z 1565.479,A 0.000,B 0.000,C 90.000,E1 122.133} C_DIS
LIN {X 0.087,Y -430.186,Z 1565.469,A 0.000,B 0.000,C 90.000,E1 120.463} C_DIS
LIN {X 0.086,Y -431.107,Z 1565.468,A 0.000,B 0.000,C 90.000,E1 120.129} C_DIS
LIN {X 0.032,Y -440.207,Z 1565.447,A 0.000,B 0.000,C 90.000,E1 116.488} C_DIS
LIN {X 0.039,Y -444.962,Z 1565.438,A 0.000,B 0.000,C 90.000,E1 114.847} C_DIS
LIN {X 0.101,Y -447.621,Z 1565.431,A 0.000,B 0.000,C 90.000,E1 113.590} C_DIS
LIN {X 0.076,Y -548.602,Z 1565.431,A 0.000,B 0.000,C 90.000,E1 113.590} C_DIS
LIN {X -0.180,Y -549.464,Z 1565.431,A 0.000,B 0.000,C 90.000,E1 113.567} C_DIS
LIN {X -0.234,Y -550.704,Z 1565.430,A 0.000,B 0.000,C 90.000,E1 113.387} C_DIS
LIN {X 0.031,Y -551.696,Z 1565.428,A 0.000,B 0.000,C 90.000,E1 113.078} C_DIS
LIN {X 0.067,Y -553.069,Z 1565.425,A 0.000,B 0.000,C 90.000,E1 112.514} C_DIS
LIN {X -0.096,Y -554.127,Z 1565.422,A 0.000,B 0.000,C 90.000,E1 111.972} C_DIS
LIN {X 0.013,Y -555.483,Z 1565.416,A 0.000,B 0.000,C 90.000,E1 110.844} C_DIS
LIN {X -0.258,Y -556.432,Z 1565.410,A 0.000,B 0.000,C 90.000,E1 109.758} C_DIS
LIN {X -0.215,Y -557.216,Z 1565.402,A 0.000,B 0.000,C 90.000,E1 108.362} C_DIS
LIN {X 0.077,Y -557.629,Z 1565.396,A 0.000,B 0.000,C 90.000,E1 107.221} C_DIS
LIN {X -0.034,Y -558.042,Z 1565.388,A 0.000,B 0.000,C 90.000,E1 105.843} C_DIS
LIN {X -0.013,Y -558.327,Z 1565.379,A 0.000,B 0.000,C 90.000,E1 104.175} C_DIS
LIN {X -0.259,Y -558.556,Z 1565.370,A 0.000,B 0.000,C 90.000,E1 102.535} C_DIS
LIN {X 0.057,Y -558.875,Z 1565.360,A 0.000,B 0.000,C 90.000,E1 100.838} C_DIS
LIN {X 0.010,Y -559.456,Z 1565.348,A 0.000,B 0.000,C 90.000,E1 98.624} C_DIS
LIN {X 0.148,Y -559.874,Z 1565.339,A 0.000,B 0.000,C 90.000,E1 96.947} C_DIS
LIN {X -0.033,Y -560.454,Z 1565.325,A 0.000,B 0.000,C 90.000,E1 94.473} C_DIS
LIN {X 0.199,Y -560.944,Z 1565.313,A 0.000,B 0.000,C 90.000,E1 92.236} C_DIS
LIN {X -0.135,Y -561.545,Z 1565.300,A 0.000,B 0.000,C 90.000,E1 90.057} C_DIS
LIN {X -0.204,Y -561.824,Z 1565.293,A 0.000,B 0.000,C 90.000,E1 88.682} C_DIS
LIN {X 0.066,Y -562.521,Z 1565.280,A 0.000,B 0.000,C 90.000,E1 86.445} C_DIS
LIN {X -0.255,Y -563.365,Z 1565.270,A 0.000,B 0.000,C 90.000,E1 84.546} C_DIS
LIN {X 0.154,Y -564.407,Z 1565.257,A 0.000,B 0.000,C 90.000,E1 82.299} C_DIS
LIN {X -0.207,Y -565.918,Z 1565.244,A 0.000,B 0.000,C 90.000,E1 79.859} C_DIS
LIN {X 0.165,Y -567.255,Z 1565.234,A 0.000,B 0.000,C 90.000,E1 78.173} C_DIS
LIN {X -0.130,Y -568.638,Z 1565.224,A 0.000,B 0.000,C 90.000,E1 76.284} C_DIS
LIN {X 0.163,Y -569.850,Z 1565.213,A 0.000,B 0.000,C 90.000,E1 74.338} C_DIS
LIN {X -0.103,Y -570.888,Z 1565.204,A 0.000,B 0.000,C 90.000,E1 72.725} C_DIS
LIN {X 0.178,Y -571.923,Z 1565.193,A 0.000,B 0.000,C 90.000,E1 70.786} C_DIS
LIN {X 0.306,Y -573.153,Z 1565.181,A 0.000,B 0.000,C 90.000,E1 68.592} C_DIS
LIN {X 0.316,Y -573.876,Z 1565.174,A 0.000,B 0.000,C 90.000,E1 67.230} C_DIS
LIN {X -0.032,Y -574.317,Z 1565.168,A 0.000,B 0.000,C 90.000,E1 66.177} C_DIS
LIN {X -0.143,Y -574.622,Z 1565.162,A 0.000,B 0.000,C 90.000,E1 65.101} C_DIS
LIN {X -0.249,Y -574.381,Z 1565.156,A 0.000,B 0.000,C 90.000,E1 64.024} C_DIS
LIN {X 0.054,Y -574.022,Z 1565.151,A 0.000,B 0.000,C 90.000,E1 63.179} C_DIS
LIN {X 0.252,Y -573.499,Z 1565.148,A 0.000,B 0.000,C 90.000,E1 62.615} C_DIS
LIN {X 0.092,Y -573.086,Z 1565.146,A 0.000,B 0.000,C 90.000,E1 62.359} C_DIS
LIN {X -0.068,Y -572.509,Z 1565.145,A 0.000,B 0.000,C 90.000,E1 62.103} C_DIS
LIN {X 0.248,Y -571.340,Z 1565.143,A 0.000,B 0.000,C 90.000,E1 61.769} C_DIS
LIN {X 0.178,Y -570.886,Z 1565.143,A 0.000,B 0.000,C 90.000,E1 61.719} C_DIS
LIN {X 0.024,Y -570.116,Z 1565.143,A 0.000,B 0.000,C 90.000,E1 61.691} C_DIS
LIN {X -0.005,Y -454.974,Z 1565.143,A 0.000,B 0.000,C 90.000,E1 61.691} C_DIS
LIN {X 0.113,Y -446.083,Z 1565.120,A 0.000,B 0.000,C 90.000,E1 57.661} C_DIS
LIN {X -0.009,Y -443.653,Z 1565.113,A 0.000,B 0.000,C 90.000,E1 56.373} C_DIS
LIN {X -0.018,Y -434.543,Z 1565.091,A 0.000,B 0.000,C 90.000,E1 52.431} C_DIS
LIN {X -0.250,Y -431.410,Z 1565.082,A 0.000,B 0.000,C 90.000,E1 50.803} C_DIS
LIN {X -0.048,Y -421.534,Z 1565.058,A 0.000,B 0.000,C 90.000,E1 46.419} C_DIS
LIN {X 0.017,Y -418.402,Z 1565.048,A 0.000,B 0.000,C 90.000,E1 44.717} C_DIS
LIN {X 0.123,Y -408.879,Z 1565.024,A 0.000,B 0.000,C 90.000,E1 40.253} C_DIS
LIN {X -0.010,Y -405.960,Z 1565.014,A 0.000,B 0.000,C 90.000,E1 38.543} C_DIS
LIN {X 0.206,Y -397.646,Z 1564.991,A 0.000,B 0.000,C 90.000,E1 34.326} C_DIS
LIN {X 0.071,Y -393.870,Z 1564.977,A 0.000,B 0.000,C 90.000,E1 31.878} C_DIS
LIN {X -0.151,Y -386.456,Z 1564.953,A 0.000,B 0.000,C 90.000,E1 27.641} C_DIS
LIN {X -0.174,Y -382.764,Z 1564.938,A 0.000,B 0.000,C 90.000,E1 24.771} C_DIS
LIN {X -0.218,Y -376.080,Z 1564.911,A 0.000,B 0.000,C 90.000,E1 20.066} C_DIS
LIN {X 0.123,Y -373.614,Z 1564.897,A 0.000,B 0.000,C 90.000,E1 17.457} C_DIS
LIN {X 0.157,Y -368.017,Z 1564.869,A 0.000,B 0.000,C 90.000,E1 12.299} C_DIS
LIN {X 0.110,Y -366.577,Z 1564.856,A 0.000,B 0.000,C 90.000,E1 10.084} C_DIS
LIN {X 0.030,Y -366.307,Z 1564.854,A 0.000,B 0.000,C 90.000,E1 9.726} C_DIS
LIN {X -0.091,Y -361.703,Z 1564.821,A 0.000,B 0.000,C 90.000,E1 3.784} C_DIS
LIN {X -0.010,Y -360.909,Z 1564.802,A 0.000,B 0.000,C 90.000,E1 0.401} C_DIS
LIN {X 0.137,Y -360.684,Z 1564.799,A 0.000,B 0.000,C 90.000,E1 359.771} C_DIS
LIN {X -0.053,Y -359.426,Z 1564.770,A 0.000,B 0.000,C 90.000,E1 354.546} C_DIS
LIN {X 0.070,Y -358.890,Z 1564.759,A 0.000,B 0.000,C 90.000,E1 352.648} C_DIS
LIN {X -0.020,Y -359.563,Z 1564.726,A 0.000,B 0.000,C 90.000,E1 346.645} C_DIS
LIN {X 0.001,Y -361.801,Z 1564.684,A 0.000,B 0.000,C 90.000,E1 339.135} C_DIS
LIN {X -0.154,Y -362.053,Z 1564.680,A 0.000,B 0.000,C 90.000,E1 338.411} C_DIS
LIN {X 0.189,Y -365.980,Z 1564.643,A 0.000,B 0.000,C 90.000,E1 331.641} C_DIS
LIN {X 0.029,Y -366.387,Z 1564.639,A 0.000,B 0.000,C 90.000,E1 330.923} C_DIS
LIN {X -0.031,Y -371.355,Z 1564.604,A 0.000,B 0.000,C 90.000,E1 324.642} C_DIS
LIN {X -0.043,Y -371.766,Z 1564.602,A 0.000,B 0.000,C 90.000,E1 324.276} C_DIS
LIN {X 0.013,Y -377.358,Z 1564.567,A 0.000,B 0.000,C 90.000,E1 318.038} C_DIS
LIN {X 0.012,Y -378.235,Z 1564.563,A 0.000,B 0.000,C 90.000,E1 317.310} C_DIS
LIN {X 0.002,Y -383.940,Z 1564.531,A 0.000,B 0.000,C 90.000,E1 311.515} C_DIS
LIN {X 0.088,Y -384.893,Z 1564.527,A 0.000,B 0.000,C 90.000,E1 310.782} C_DIS
LIN {X 0.262,Y -390.610,Z 1564.495,A 0.000,B 0.000,C 90.000,E1 305.025} C_DIS
LIN {X 0.106,Y -391.104,Z 1564.493,A 0.000,B 0.000,C 90.000,E1 304.692} C_DIS
LIN {X 0.022,Y -391.648,Z 1564.489,A 0.000,B 0.000,C 90.000,E1 303.992} C_DIS
LIN {X -0.080,Y -396.825,Z 1564.459,A 0.000,B 0.000,C 90.000,E1 298.693} C_DIS
LIN {X -0.210,Y -397.120,Z 1564.457,A 0.000,B 0.000,C 90.000,E1 298.359} C_DIS
LIN {X -0.055,Y -401.597,Z 1564.426,A 0.000,B 0.000,C 90.000,E1 292.717} C_DIS
LIN {X 0.222,Y -404.659,Z 1564.395,A 0.000,B 0.000,C 90.000,E1 287.094} C_DIS
LIN {X -0.079,Y -404.735,Z 1564.391,A 0.000,B 0.000,C 90.000,E1 286.441} C_DIS
LIN {X 0.214,Y -406.099,Z 1564.364,A 0.000,B 0.000,C 90.000,E1 281.535} C_DIS
LIN {X -0.176,Y -406.094,Z 1564.362,A 0.000,B 0.000,C 90.000,E1 281.243} C_DIS
LIN {X -0.097,Y -405.680,Z 1564.333,A 0.000,B 0.000,C 90.000,E1 276.024} C_DIS
LIN {X -0.165,Y -405.058,Z 1564.328,A 0.000,B 0.000,C 90.000,E1 274.992} C_DIS
LIN {X -0.060,Y -403.497,Z 1564.304,A 0.000,B 0.000,C 90.000,E1 270.802} C_DIS
LIN {X -0.092,Y -403.288,Z 1564.302,A 0.000,B 0.000,C 90.000,E1 270.458} C_DIS
LIN {X 0.091,Y -398.931,Z 1564.271,A 0.000,B 0.000,C 90.000,E1 264.837} C_DIS
LIN {X -0.040,Y -393.108,Z 1564.242,A 0.000,B 0.000,C 90.000,E1 259.567} C_DIS
LIN {X -0.079,Y -392.835,Z 1564.240,A 0.000,B 0.000,C 90.000,E1 259.218} C_DIS
LIN {X 0.034,Y -385.993,Z 1564.212,A 0.000,B 0.000,C 90.000,E1 254.212} C_DIS
LIN {X -0.026,Y -385.267,Z 1564.208,A 0.000,B 0.000,C 90.000,E1 253.504} C_DIS
LIN {X -0.004,Y -384.768,Z 1564.206,A 0.000,B 0.000,C 90.000,E1 253.142} C_DIS
LIN {X 0.221,Y -377.973,Z 1564.182,A 0.000,B 0.000,C 90.000,E1 248.773} C_DIS
LIN {X -0.044,Y -376.233,Z 1564.174,A 0.000,B 0.000,C 90.000,E1 247.358} C_DIS
LIN {X 0.057,Y -374.944,Z 1564.170,A 0.000,B 0.000,C 90.000,E1 246.613} C_DIS
LIN {X -0.208,Y -368.417,Z 1564.148,A 0.000,B 0.000,C 90.000,E1 242.615} C_DIS
LIN {X 0.097,Y -366.047,Z 1564.137,A 0.000,B 0.000,C 90.000,E1 240.717} C_DIS
LIN {X 0.004,Y -359.196,Z 1564.115,A 0.000,B 0.000,C 90.000,E1 236.628} C_DIS
LIN {X 0.021,Y -355.842,Z 1564.100,A 0.000,B 0.000,C 90.000,E1 233.989} C_DIS
LIN {X -0.173,Y -348.793,Z 1564.075,A 0.000,B 0.000,C 90.000,E1 229.461} C_DIS
LIN {X -0.097,Y -346.185,Z 1564.062,A 0.000,B 0.000,C 90.000,E1 227.148} C_DIS
LIN {X -0.088,Y -345.065,Z 1564.058,A 0.000,B 0.000,C 90.000,E1 226.377} C_DIS
LIN {X 0.094,Y -338.586,Z 1564.030,A 0.000,B 0.000,C 90.000,E1 221.310} C_DIS
LIN {X 0.094,Y -336.840,Z 1564.019,A 0.000,B 0.000,C 90.000,E1 219.358} C_DIS
LIN {X 0.014,Y -330.861,Z 1563.988,A 0.000,B 0.000,C 90.000,E1 213.865} C_DIS
LIN {X 0.149,Y -329.296,Z 1563.975,A 0.000,B 0.000,C 90.000,E1 211.465} C_DIS
LIN {X -0.154,Y -324.669,Z 1563.942,A 0.000,B 0.000,C 90.000,E1 205.540} C_DIS
LIN {X 0.174,Y -323.837,Z 1563.928,A 0.000,B 0.000,C 90.000,E1 203.078} C_DIS
LIN {X -0.017,Y -321.124,Z 1563.881,A 0.000,B 0.000,C 90.000,E1 194.662} C_DIS
LIN {X 0.138,Y -320.932,Z 1563.877,A 0.000,B 0.000,C 90.000,E1 193.828} C_DIS
LIN {X -0.076,Y -321.562,Z 1563.832,A 0.000,B 0.000,C 90.000,E1 185.796} C_DIS
LIN {X -0.143,Y -324.415,Z 1563.790,A 0.000,B 0.000,C 90.000,E1 178.165} C_DIS
LIN {X -0.141,Y -325.376,Z 1563.783,A 0.000,B 0.000,C 90.000,E1 176.963} C_DIS
LIN {X -0.100,Y -329.112,Z 1563.750,A 0.000,B 0.000,C 90.000,E1 170.971} C_DIS
LIN {X 0.061,Y -334.260,Z 1563.726,A 0.000,B 0.000,C 90.000,E1 166.589} C_DIS
LIN {X 0.067,Y -335.488,Z 1563.719,A 0.000,B 0.000,C 90.000,E1 165.408} C_DIS
LIN {X 0.143,Y -340.932,Z 1563.695,A 0.000,B 0.000,C 90.000,E1 161.094} C_DIS
LIN {X -0.172,Y -342.138,Z 1563.691,A 0.000,B 0.000,C 90.000,E1 160.369} C_DIS
LIN {X -0.058,Y -347.939,Z 1563.667,A 0.000,B 0.000,C 90.000,E1 156.102} C_DIS
LIN {X -0.081,Y -354.259,Z 1563.648,A 0.000,B 0.000,C 90.000,E1 152.666} C_DIS
LIN {X -0.222,Y -361.406,Z 1563.625,A 0.000,B 0.000,C 90.000,E1 148.535} C_DIS
LIN {X 0.065,Y -368.758,Z 1563.606,A 0.000,B 0.000,C 90.000,E1 145.135} C_DIS
LIN {X 0.065,Y -377.029,Z 1563.584,A 0.000,B 0.000,C 90.000,E1 141.090} C_DIS
LIN {X -0.061,Y -383.435,Z 1563.570,A 0.000,B 0.000,C 90.000,E1 138.566} C_DIS
LIN {X -0.015,Y -385.037,Z 1563.566,A 0.000,B 0.000,C 90.000,E1 137.838} C_DIS
LIN {X -0.004,Y -394.325,Z 1563.544,A 0.000,B 0.000,C 90.000,E1 133.905} C_DIS
LIN {X 0.107,Y -399.276,Z 1563.534,A 0.000,B 0.000,C 90.000,E1 132.123} C_DIS
LIN {X 0.210,Y -400.192,Z 1563.532,A 0.000,B 0.000,C 90.000,E1 131.757} C_DIS
LIN {X -0.113,Y -409.687,Z 1563.511,A 0.000,B 0.000,C 90.000,E1 127.971} C_DIS
LIN {X 0.046,Y -415.746,Z 1563.499,A 0.000,B 0.000,C 90.000,E1 125.884} C_DIS
LIN {X 0.153,Y -425.188,Z 1563.479,A 0.000,B 0.000,C 90.000,E1 122.133} C_DIS
LIN {X 0.087,Y -430.186,Z 1563.469,A 0.000,B 0.000,C 90.000,E1 120.463} C_DIS
LIN {X 0.086,Y -431.107,Z 1563.468,A 0.000,B 0.000,C 90.000,E1 120.129} C_DIS
LIN {X 0.032,Y -440.207,Z 1563.447,A 0.000,B 0.000,C 90.000,E1 116.488} C_DIS
LIN {X -0.137,Y -443.998,Z 1563.440,A 0.000,B 0.000,C 90.000,E1 115.207} C_DIS
LIN {X -0.202,Y -548.249,Z 1563.440,A 0.000,B 0.000,C 90.000,E1 115.207} C_DIS
LIN {X 0.229,Y -548.567,Z 1563.440,A 0.000,B 0.000,C 90.000,E1 115.155} C_DIS
LIN {X 0.209,Y -549.602,Z 1563.439,A 0.000,B 0.000,C 90.000,E1 115.079} C_DIS
LIN {X -0.234,Y -550.966,Z 1563.438,A 0.000,B 0.000,C 90.000,E1 114.899} C_DIS
LIN {X 0.030,Y -551.973,Z 1563.437,A 0.000,B 0.000,C 90.000,E1 114.591} C_DIS
LIN {X 0.072,Y -553.289,Z 1563.434,A 0.000,B 0.000,C 90.000,E1 114.027} C_DIS
LIN {X 0.124,Y -554.375,Z 1563.430,A 0.000,B 0.000,C 90.000,E1 113.462} C_DIS
LIN {X 0.248,Y -555.679,Z 1563.424,A 0.000,B 0.000,C 90.000,E1 112.333} C_DIS
LIN {X 0.107,Y -556.210,Z 1563.421,A 0.000,B 0.000,C 90.000,E1 111.791} C_DIS
LIN {X 0.246,Y -556.986,Z 1563.415,A 0.000,B 0.000,C 90.000,E1 110.663} C_DIS
LIN {X -0.003,Y -557.496,Z 1563.409,A 0.000,B 0.000,C 90.000,E1 109.577} C_DIS
LIN {X 0.059,Y -557.890,Z 1563.401,A 0.000,B 0.000,C 90.000,E1 108.181} C_DIS
LIN {X -0.031,Y -558.332,Z 1563.389,A 0.000,B 0.000,C 90.000,E1 105.969} C_DIS
LIN {X 0.143,Y -558.647,Z 1563.378,A 0.000,B 0.000,C 90.000,E1 104.008} C_DIS
LIN {X 0.178,Y -558.940,Z 1563.367,A 0.000,B 0.000,C 90.000,E1 102.063} C_DIS
LIN {X -0.197,Y -559.218,Z 1563.359,A 0.000,B 0.000,C 90.000,E1 100.715} C_DIS
LIN {X 0.078,Y -559.772,Z 1563.349,A 0.000,B 0.000,C 90.000,E1 98.746} C_DIS
LIN {X 0.234,Y -560.164,Z 1563.339,A 0.000,B 0.000,C 90.000,E1 97.068} C_DIS
LIN {X -0.173,Y -560.515,Z 1563.330,A 0.000,B 0.000,C 90.000,E1 95.448} C_DIS
LIN {X -0.217,Y -560.890,Z 1563.323,A 0.000,B 0.000,C 90.000,E1 94.069} C_DIS
LIN {X -0.099,Y -561.367,Z 1563.312,A 0.000,B 0.000,C 90.000,E1 92.121} C_DIS
LIN {X 0.041,Y -561.889,Z 1563.301,A 0.000,B 0.000,C 90.000,E1 90.172} C_DIS
LIN {X -0.020,Y -562.212,Z 1563.293,A 0.000,B 0.000,C 90.000,E1 88.797} C_DIS
LIN {X 0.132,Y -562.796,Z 1563.283,A 0.000,B 0.000,C 90.000,E1 86.849} C_DIS
LIN {X -0.194,Y -563.592,Z 1563.272,A 0.000,B 0.000,C 90.000,E1 84.951} C_DIS
LIN {X 0.219,Y -564.639,Z 1563.260,A 0.000,B 0.000,C 90.000,E1 82.704} C_DIS
LIN {X -0.231,Y -566.126,Z 1563.246,A 0.000,B 0.000,C 90.000,E1 80.274} C_DIS
LIN {X 0.045,Y -567.807,Z 1563.234,A 0.000,B 0.000,C 90.000,E1 78.049} C_DIS
LIN {X 0.013,Y -569.017,Z 1563.224,A 0.000,B 0.000,C 90.000,E1 76.408} C_DIS
LIN {X 0.320,Y -569.702,Z 1563.219,A 0.000,B 0.000,C 90.000,E1 75.283} C_DIS
LIN {X -0.102,Y -570.724,Z 1563.209,A 0.000,B 0.000,C 90.000,E1 73.685} C_DIS
LIN {X -0.158,Y -571.401,Z 1563.203,A 0.000,B 0.000,C 90.000,E1 72.598} C_DIS
LIN {X -0.048,Y -572.452,Z 1563.193,A 0.000,B 0.000,C 90.000,E1 70.678} C_DIS
LIN {X -0.074,Y -573.541,Z 1563.182,A 0.000,B 0.000,C 90.000,E1 68.773} C_DIS
LIN {X -0.073,Y -574.757,Z 1563.172,A 0.000,B 0.000,C 90.000,E1 66.869} C_DIS
LIN {X 0.033,Y -575.718,Z 1563.162,A 0.000,B 0.000,C 90.000,E1 65.229} C_DIS
LIN {X 0.095,Y -575.921,Z 1563.158,A 0.000,B 0.000,C 90.000,E1 64.409} C_DIS
LIN {X 0.112,Y -576.150,Z 1563.150,A 0.000,B 0.000,C 90.000,E1 63.050} C_DIS
LIN {X 0.020,Y -575.935,Z 1563.144,A 0.000,B 0.000,C 90.000,E1 61.975} C_DIS
LIN {X -0.012,Y -575.616,Z 1563.141,A 0.000,B 0.000,C 90.000,E1 61.435} C_DIS
LIN {X -0.319,Y -574.980,Z 1563.138,A 0.000,B 0.000,C 90.000,E1 60.923} C_DIS
LIN {X 0.308,Y -574.489,Z 1563.137,A 0.000,B 0.000,C 90.000,E1 60.589} C_DIS
LIN {X 0.060,Y -573.513,Z 1563.135,A 0.000,B 0.000,C 90.000,E1 60.284} C_DIS
LIN {X 0.210,Y -572.653,Z 1563.134,A 0.000,B 0.000,C 90.000,E1 60.127} C_DIS
LIN {X -0.272,Y -572.065,Z 1563.134,A 0.000,B 0.000,C 90.000,E1 60.127} C_DIS
LIN {X 0.107,Y -571.777,Z 1563.134,A 0.000,B 0.000,C 90.000,E1 60.078} C_DIS
LIN {X 0.038,Y -451.099,Z 1563.134,A 0.000,B 0.000,C 90.000,E1 60.078} C_DIS
LIN {X -0.015,Y -444.318,Z 1563.115,A 0.000,B 0.000,C 90.000,E1 56.707} C_DIS
LIN {X 0.043,Y -443.670,Z 1563.113,A 0.000,B 0.000,C 90.000,E1 56.373} C_DIS
LIN {X 0.033,Y -434.556,Z 1563.091,A 0.000,B 0.000,C 90.000,E1 52.431} C_DIS
LIN {X -0.198,Y -431.426,Z 1563.082,A 0.000,B 0.000,C 90.000,E1 50.803} C_DIS
LIN {X 0.003,Y -421.547,Z 1563.058,A 0.000,B 0.000,C 90.000,E1 46.419} C_DIS
LIN {X -0.226,Y -418.420,Z 1563.049,A 0.000,B 0.000,C 90.000,E1 44.757} C_DIS
LIN {X 0.174,Y -408.892,Z 1563.024,A 0.000,B 0.000,C 90.000,E1 40.253} C_DIS
LIN {X 0.040,Y -405.971,Z 1563.014,A 0.000,B 0.000,C 90.000,E1 38.543} C_DIS
LIN {X 0.032,Y -397.658,Z 1562.991,A 0.000,B 0.000,C 90.000,E1 34.358} C_DIS
LIN {X 0.122,Y -393.880,Z 1562.977,A 0.000,B 0.000,C 90.000,E1 31.878} C_DIS
LIN {X -0.101,Y -386.467,Z 1562.953,A 0.000,B 0.000,C 90.000,E1 27.641} C_DIS
LIN {X -0.124,Y -382.776,Z 1562.938,A 0.000,B 0.000,C 90.000,E1 24.771} C_DIS
LIN {X -0.169,Y -376.088,Z 1562.911,A 0.000,B 0.000,C 90.000,E1 20.066} C_DIS
LIN {X 0.173,Y -373.621,Z 1562.897,A 0.000,B 0.000,C 90.000,E1 17.457} C_DIS
LIN {X -0.153,Y -368.022,Z 1562.869,A 0.000,B 0.000,C 90.000,E1 12.355} C_DIS
LIN {X 0.078,Y -366.315,Z 1562.854,A 0.000,B 0.000,C 90.000,E1 9.726} C_DIS
LIN {X -0.043,Y -361.707,Z 1562.821,A 0.000,B 0.000,C 90.000,E1 3.784} C_DIS
LIN {X 0.038,Y -360.909,Z 1562.802,A 0.000,B 0.000,C 90.000,E1 0.401} C_DIS
LIN {X 0.137,Y -360.684,Z 1562.799,A 0.000,B 0.000,C 90.000,E1 359.771} C_DIS
LIN {X -0.053,Y -359.426,Z 1562.770,A 0.000,B 0.000,C 90.000,E1 354.546} C_DIS
LIN {X 0.070,Y -358.890,Z 1562.759,A 0.000,B 0.000,C 90.000,E1 352.648} C_DIS
LIN {X -0.020,Y -359.563,Z 1562.726,A 0.000,B 0.000,C 90.000,E1 346.645} C_DIS
LIN {X 0.001,Y -361.801,Z 1562.684,A 0.000,B 0.000,C 90.000,E1 339.135} C_DIS
LIN {X -0.154,Y -362.053,Z 1562.680,A 0.000,B 0.000,C 90.000,E1 338.411} C_DIS
LIN {X 0.189,Y -365.980,Z 1562.643,A 0.000,B 0.000,C 90.000,E1 331.641} C_DIS
LIN {X 0.029,Y -366.387,Z 1562.639,A 0.000,B 0.000,C 90.000,E1 330.923} C_DIS
LIN {X -0.031,Y -371.355,Z 1562.604,A 0.000,B 0.000,C 90.000,E1 324.642} C_DIS
LIN {X -0.043,Y -371.766,Z 1562.602,A 0.000,B 0.000,C 90.000,E1 324.276} C_DIS
LIN {X 0.013,Y -377.358,Z 1562.567,A 0.000,B 0.000,C 90.000,E1 318.038} C_DIS
LIN {X 0.012,Y -378.235,Z 1562.563,A 0.000,B 0.000,C 90.000,E1 317.310} C_DIS
LIN {X 0.002,Y -383.940,Z 1562.531,A 0.000,B 0.000,C 90.000,E1 311.515} C_DIS
LIN {X 0.088,Y -384.893,Z 1562.527,A 0.000,B 0.000,C 90.000,E1 310.782} C_DIS
LIN {X 0.262,Y -390.610,Z 1562.495,A 0.000,B 0.000,C 90.000,E1 305.025} C_DIS
LIN {X 0.106,Y -391.104,Z 1562.493,A 0.000,B 0.000,C 90.000,E1 304.692} C_DIS
LIN {X 0.022,Y -391.648,Z 1562.489,A 0.000,B 0.000,C 90.000,E1 303.992} C_DIS
LIN {X -0.080,Y -396.825,Z 1562.459,A 0.000,B 0.000,C 90.000,E1 298.693} C_DIS
LIN {X -0.210,Y -397.120,Z 1562.457,A 0.000,B 0.000,C 90.000,E1 298.359} C_DIS
LIN {X -0.055,Y -401.597,Z 1562.426,A 0.000,B 0.000,C 90.000,E1 292.717} C_DIS
LIN {X 0.222,Y -404.659,Z 1562.395,A 0.000,B 0.000,C 90.000,E1 287.094} C_DIS
LIN {X -0.079,Y -404.735,Z 1562.391,A 0.000,B 0.000,C 90.000,E1 286.441} C_DIS
LIN {X 0.214,Y -406.099,Z 1562.364,A 0.000,B 0.000,C 90.000,E1 281.535} C_DIS
LIN {X -0.176,Y -406.094,Z 1562.362,A 0.000,B 0.000,C 90.000,E1 281.243} C_DIS
LIN {X -0.097,Y -405.680,Z 1562.333,A 0.000,B 0.000,C 90.000,E1 276.024} C_DIS
LIN {X -0.165,Y -405.058,Z 1562.328,A 0.000,B 0.000,C 90.000,E1 274.992} C_DIS
LIN {X -0.060,Y -403.497,Z 1562.304,A 0.000,B 0.000,C 90.000,E1 270.802} C_DIS
LIN {X -0.092,Y -403.288,Z 1562.302,A 0.000,B 0.000,C 90.000,E1 270.458} C_DIS
LIN {X 0.091,Y -398.931,Z 1562.271,A 0.000,B 0.000,C 90.000,E1 264.837} C_DIS
LIN {X -0.040,Y -393.108,Z 1562.242,A 0.000,B 0.000,C 90.000,E1 259.567} C_DIS
LIN {X -0.079,Y -392.835,Z 1562.240,A 0.000,B 0.000,C 90.000,E1 259.218} C_DIS
LIN {X 0.034,Y -385.993,Z 1562.212,A 0.000,B 0.000,C 90.000,E1 254.212} C_DIS
LIN {X -0.026,Y -385.267,Z 1562.208,A 0.000,B 0.000,C 90.000,E1 253.504} C_DIS
LIN {X -0.004,Y -384.768,Z 1562.206,A 0.000,B 0.000,C 90.000,E1 253.142} C_DIS
LIN {X 0.221,Y -377.973,Z 1562.182,A 0.000,B 0.000,C 90.000,E1 248.773} C_DIS
LIN {X -0.044,Y -376.233,Z 1562.174,A 0.000,B 0.000,C 90.000,E1 247.358} C_DIS
LIN {X 0.057,Y -374.944,Z 1562.170,A 0.000,B 0.000,C 90.000,E1 246.613} C_DIS
LIN {X -0.208,Y -368.417,Z 1562.148,A 0.000,B 0.000,C 90.000,E1 242.615} C_DIS
LIN {X 0.097,Y -366.047,Z 1562.137,A 0.000,B 0.000,C 90.000,E1 240.717} C_DIS
LIN {X 0.004,Y -359.196,Z 1562.115,A 0.000,B 0.000,C 90.000,E1 236.628} C_DIS
LIN {X 0.021,Y -355.842,Z 1562.100,A 0.000,B 0.000,C 90.000,E1 233.989} C_DIS
LIN {X -0.173,Y -348.793,Z 1562.075,A 0.000,B 0.000,C 90.000,E1 229.461} C_DIS
LIN {X -0.097,Y -346.185,Z 1562.062,A 0.000,B 0.000,C 90.000,E1 227.148} C_DIS
LIN {X -0.088,Y -345.065,Z 1562.058,A 0.000,B 0.000,C 90.000,E1 226.377} C_DIS
LIN {X 0.094,Y -338.586,Z 1562.030,A 0.000,B 0.000,C 90.000,E1 221.310} C_DIS
LIN {X 0.094,Y -336.840,Z 1562.019,A 0.000,B 0.000,C 90.000,E1 219.358} C_DIS
LIN {X 0.014,Y -330.861,Z 1561.988,A 0.000,B 0.000,C 90.000,E1 213.865} C_DIS
LIN {X 0.149,Y -329.296,Z 1561.975,A 0.000,B 0.000,C 90.000,E1 211.465} C_DIS
LIN {X -0.154,Y -324.669,Z 1561.942,A 0.000,B 0.000,C 90.000,E1 205.540} C_DIS
LIN {X 0.174,Y -323.837,Z 1561.928,A 0.000,B 0.000,C 90.000,E1 203.078} C_DIS
LIN {X -0.017,Y -321.124,Z 1561.881,A 0.000,B 0.000,C 90.000,E1 194.662} C_DIS
LIN {X 0.138,Y -320.932,Z 1561.877,A 0.000,B 0.000,C 90.000,E1 193.828} C_DIS
LIN {X -0.076,Y -321.562,Z 1561.832,A 0.000,B 0.000,C 90.000,E1 185.796} C_DIS
LIN {X -0.143,Y -324.415,Z 1561.790,A 0.000,B 0.000,C 90.000,E1 178.165} C_DIS
LIN {X -0.141,Y -325.376,Z 1561.783,A 0.000,B 0.000,C 90.000,E1 176.963} C_DIS
LIN {X -0.100,Y -329.112,Z 1561.750,A 0.000,B 0.000,C 90.000,E1 170.971} C_DIS
LIN {X 0.061,Y -334.260,Z 1561.726,A 0.000,B 0.000,C 90.000,E1 166.589} C_DIS
LIN {X 0.067,Y -335.488,Z 1561.719,A 0.000,B 0.000,C 90.000,E1 165.408} C_DIS
LIN {X 0.143,Y -340.932,Z 1561.695,A 0.000,B 0.000,C 90.000,E1 161.094} C_DIS
LIN {X -0.172,Y -342.138,Z 1561.691,A 0.000,B 0.000,C 90.000,E1 160.369} C_DIS
LIN {X -0.058,Y -347.939,Z 1561.667,A 0.000,B 0.000,C 90.000,E1 156.102} C_DIS
LIN {X -0.081,Y -354.259,Z 1561.648,A 0.000,B 0.000,C 90.000,E1 152.666} C_DIS
LIN {X -0.222,Y -361.406,Z 1561.625,A 0.000,B 0.000,C 90.000,E1 148.535} C_DIS
LIN {X 0.065,Y -368.758,Z 1561.606,A 0.000,B 0.000,C 90.000,E1 145.135} C_DIS
LIN {X 0.065,Y -377.029,Z 1561.584,A 0.000,B 0.000,C 90.000,E1 141.090} C_DIS
LIN {X -0.061,Y -383.435,Z 1561.570,A 0.000,B 0.000,C 90.000,E1 138.566} C_DIS
LIN {X -0.015,Y -385.037,Z 1561.566,A 0.000,B 0.000,C 90.000,E1 137.838} C_DIS
LIN {X -0.004,Y -394.325,Z 1561.544,A 0.000,B 0.000,C 90.000,E1 133.905} C_DIS
LIN {X 0.107,Y -399.276,Z 1561.534,A 0.000,B 0.000,C 90.000,E1 132.123} C_DIS
LIN {X 0.210,Y -400.192,Z 1561.532,A 0.000,B 0.000,C 90.000,E1 131.757} C_DIS
LIN {X -0.113,Y -409.687,Z 1561.511,A 0.000,B 0.000,C 90.000,E1 127.971} C_DIS
LIN {X 0.046,Y -415.746,Z 1561.499,A 0.000,B 0.000,C 90.000,E1 125.884} C_DIS
LIN {X 0.153,Y -425.188,Z 1561.479,A 0.000,B 0.000,C 90.000,E1 122.133} C_DIS
LIN {X 0.087,Y -430.186,Z 1561.469,A 0.000,B 0.000,C 90.000,E1 120.463} C_DIS
LIN {X 0.086,Y -431.107,Z 1561.468,A 0.000,B 0.000,C 90.000,E1 120.129} C_DIS
LIN {X 0.073,Y -439.693,Z 1561.448,A 0.000,B 0.000,C 90.000,E1 116.668} C_DIS
LIN {X 0.045,Y -547.980,Z 1561.448,A 0.000,B 0.000,C 90.000,E1 116.668} C_DIS
LIN {X -0.047,Y -548.405,Z 1561.448,A 0.000,B 0.000,C 90.000,E1 116.668} C_DIS
LIN {X 0.040,Y -550.082,Z 1561.447,A 0.000,B 0.000,C 90.000,E1 116.488} C_DIS
LIN {X -0.076,Y -551.346,Z 1561.446,A 0.000,B 0.000,C 90.000,E1 116.232} C_DIS
LIN {X 0.186,Y -552.258,Z 1561.444,A 0.000,B 0.000,C 90.000,E1 115.924} C_DIS
LIN {X -0.044,Y -553.000,Z 1561.443,A 0.000,B 0.000,C 90.000,E1 115.668} C_DIS
LIN {X 0.015,Y -554.600,Z 1561.438,A 0.000,B 0.000,C 90.000,E1 114.823} C_DIS
LIN {X -0.148,Y -555.613,Z 1561.433,A 0.000,B 0.000,C 90.000,E1 114.003} C_DIS
LIN {X -0.083,Y -556.248,Z 1561.430,A 0.000,B 0.000,C 90.000,E1 113.439} C_DIS
LIN {X 0.141,Y -557.178,Z 1561.422,A 0.000,B 0.000,C 90.000,E1 112.025} C_DIS
LIN {X -0.134,Y -557.722,Z 1561.415,A 0.000,B 0.000,C 90.000,E1 110.663} C_DIS
LIN {X -0.076,Y -557.981,Z 1561.407,A 0.000,B 0.000,C 90.000,E1 109.268} C_DIS
LIN {X -0.010,Y -558.241,Z 1561.399,A 0.000,B 0.000,C 90.000,E1 107.873} C_DIS
LIN {X 0.305,Y -558.627,Z 1561.389,A 0.000,B 0.000,C 90.000,E1 105.898} C_DIS
LIN {X 0.195,Y -558.861,Z 1561.379,A 0.000,B 0.000,C 90.000,E1 104.245} C_DIS
LIN {X 0.095,Y -559.157,Z 1561.370,A 0.000,B 0.000,C 90.000,E1 102.591} C_DIS
LIN {X 0.017,Y -559.535,Z 1561.359,A 0.000,B 0.000,C 90.000,E1 100.658} C_DIS
LIN {X -0.249,Y -560.108,Z 1561.349,A 0.000,B 0.000,C 90.000,E1 98.746} C_DIS
LIN {X -0.158,Y -560.424,Z 1561.341,A 0.000,B 0.000,C 90.000,E1 97.352} C_DIS
LIN {X 0.072,Y -560.889,Z 1561.330,A 0.000,B 0.000,C 90.000,E1 95.391} C_DIS
LIN {X 0.036,Y -561.279,Z 1561.322,A 0.000,B 0.000,C 90.000,E1 94.012} C_DIS
LIN {X 0.166,Y -561.763,Z 1561.312,A 0.000,B 0.000,C 90.000,E1 92.064} C_DIS
LIN {X -0.246,Y -562.283,Z 1561.301,A 0.000,B 0.000,C 90.000,E1 90.172} C_DIS
LIN {X 0.261,Y -562.636,Z 1561.293,A 0.000,B 0.000,C 90.000,E1 88.740} C_DIS
LIN {X -0.107,Y -563.234,Z 1561.282,A 0.000,B 0.000,C 90.000,E1 86.846} C_DIS
LIN {X 0.108,Y -564.030,Z 1561.272,A 0.000,B 0.000,C 90.000,E1 84.894} C_DIS
LIN {X -0.028,Y -565.087,Z 1561.260,A 0.000,B 0.000,C 90.000,E1 82.704} C_DIS
LIN {X 0.016,Y -566.399,Z 1561.247,A 0.000,B 0.000,C 90.000,E1 80.500} C_DIS
LIN {X -0.175,Y -568.268,Z 1561.234,A 0.000,B 0.000,C 90.000,E1 78.049} C_DIS
LIN {X 0.173,Y -569.301,Z 1561.226,A 0.000,B 0.000,C 90.000,E1 76.645} C_DIS
LIN {X 0.116,Y -570.218,Z 1561.218,A 0.000,B 0.000,C 90.000,E1 75.283} C_DIS
LIN {X 0.222,Y -571.531,Z 1561.206,A 0.000,B 0.000,C 90.000,E1 73.087} C_DIS
LIN {X -0.192,Y -572.258,Z 1561.199,A 0.000,B 0.000,C 90.000,E1 71.764} C_DIS
LIN {X 0.133,Y -573.077,Z 1561.191,A 0.000,B 0.000,C 90.000,E1 70.369} C_DIS
LIN {X -0.241,Y -574.022,Z 1561.182,A 0.000,B 0.000,C 90.000,E1 68.773} C_DIS
LIN {X 0.157,Y -575.037,Z 1561.173,A 0.000,B 0.000,C 90.000,E1 67.102} C_DIS
LIN {X 0.195,Y -575.939,Z 1561.165,A 0.000,B 0.000,C 90.000,E1 65.741} C_DIS
LIN {X -0.265,Y -576.488,Z 1561.161,A 0.000,B 0.000,C 90.000,E1 64.973} C_DIS
LIN {X -0.011,Y -577.409,Z 1561.150,A 0.000,B 0.000,C 90.000,E1 63.050} C_DIS
LIN {X 0.041,Y -577.761,Z 1561.143,A 0.000,B 0.000,C 90.000,E1 61.691} C_DIS
LIN {X 0.105,Y -577.678,Z 1561.138,A 0.000,B 0.000,C 90.000,E1 60.873} C_DIS
LIN {X 0.090,Y -577.498,Z 1561.135,A 0.000,B 0.000,C 90.000,E1 60.333} C_DIS
LIN {X 0.078,Y -577.028,Z 1561.132,A 0.000,B 0.000,C 90.000,E1 59.793} C_DIS
LIN {X 0.065,Y -576.174,Z 1561.129,A 0.000,B 0.000,C 90.000,E1 59.253} C_DIS
LIN {X -0.090,Y -575.506,Z 1561.128,A 0.000,B 0.000,C 90.000,E1 58.997} C_DIS
LIN {X 0.244,Y -574.166,Z 1561.126,A 0.000,B 0.000,C 90.000,E1 58.663} C_DIS
LIN {X 0.157,Y -573.619,Z 1561.126,A 0.000,B 0.000,C 90.000,E1 58.614} C_DIS
LIN {X -0.162,Y -572.920,Z 1561.126,A 0.000,B 0.000,C 90.000,E1 58.614} C_DIS
LIN {X 0.063,Y -447.886,Z 1561.126,A 0.000,B 0.000,C 90.000,E1 58.584} C_DIS
LIN {X -0.054,Y -443.945,Z 1561.114,A 0.000,B 0.000,C 90.000,E1 56.501} C_DIS
LIN {X 0.232,Y -434.131,Z 1561.090,A 0.000,B 0.000,C 90.000,E1 52.190} C_DIS
LIN {X 0.074,Y -431.653,Z 1561.083,A 0.000,B 0.000,C 90.000,E1 50.884} C_DIS
LIN {X -0.069,Y -426.026,Z 1561.070,A 0.000,B 0.000,C 90.000,E1 48.566} C_DIS
LIN {X 0.052,Y -418.684,Z 1561.049,A 0.000,B 0.000,C 90.000,E1 44.838} C_DIS
LIN {X -0.009,Y -409.751,Z 1561.026,A 0.000,B 0.000,C 90.000,E1 40.744} C_DIS
LIN {X 0.015,Y -406.163,Z 1561.015,A 0.000,B 0.000,C 90.000,E1 38.669} C_DIS
LIN {X 0.048,Y -404.727,Z 1561.011,A 0.000,B 0.000,C 90.000,E1 37.971} C_DIS
LIN {X 0.076,Y -396.134,Z 1560.986,A 0.000,B 0.000,C 90.000,E1 33.420} C_DIS
LIN {X 0.098,Y -394.050,Z 1560.978,A 0.000,B 0.000,C 90.000,E1 32.005} C_DIS
LIN {X -0.173,Y -392.769,Z 1560.974,A 0.000,B 0.000,C 90.000,E1 31.337} C_DIS
LIN {X 0.062,Y -385.138,Z 1560.948,A 0.000,B 0.000,C 90.000,E1 26.668} C_DIS
LIN {X -0.135,Y -382.939,Z 1560.938,A 0.000,B 0.000,C 90.000,E1 24.899} C_DIS
LIN {X -0.036,Y -376.232,Z 1560.912,A 0.000,B 0.000,C 90.000,E1 20.174} C_DIS
LIN {X -0.171,Y -373.729,Z 1560.898,A 0.000,B 0.000,C 90.000,E1 17.638} C_DIS
LIN {X 0.072,Y -371.868,Z 1560.890,A 0.000,B 0.000,C 90.000,E1 16.134} C_DIS
LIN {X 0.050,Y -366.856,Z 1560.859,A 0.000,B 0.000,C 90.000,E1 10.602} C_DIS
LIN {X 0.127,Y -366.450,Z 1560.855,A 0.000,B 0.000,C 90.000,E1 9.849} C_DIS
LIN {X 0.064,Y -361.763,Z 1560.822,A 0.000,B 0.000,C 90.000,E1 3.898} C_DIS
LIN {X -0.050,Y -360.887,Z 1560.801,A 0.000,B 0.000,C 90.000,E1 0.172} C_DIS
LIN {X -0.053,Y -359.426,Z 1560.770,A 0.000,B 0.000,C 90.000,E1 354.546} C_DIS
LIN {X 0.070,Y -358.890,Z 1560.759,A 0.000,B 0.000,C 90.000,E1 352.648} C_DIS
LIN {X -0.020,Y -359.563,Z 1560.726,A 0.000,B 0.000,C 90.000,E1 346.645} C_DIS
LIN {X 0.001,Y -361.801,Z 1560.684,A 0.000,B 0.000,C 90.000,E1 339.135} C_DIS
LIN {X -0.154,Y -362.053,Z 1560.680,A 0.000,B 0.000,C 90.000,E1 338.411} C_DIS
LIN {X 0.189,Y -365.980,Z 1560.643,A 0.000,B 0.000,C 90.000,E1 331.641} C_DIS
LIN {X 0.029,Y -366.387,Z 1560.639,A 0.000,B 0.000,C 90.000,E1 330.923} C_DIS
LIN {X -0.031,Y -371.355,Z 1560.604,A 0.000,B 0.000,C 90.000,E1 324.642} C_DIS
LIN {X -0.043,Y -371.766,Z 1560.602,A 0.000,B 0.000,C 90.000,E1 324.276} C_DIS
LIN {X 0.013,Y -377.358,Z 1560.567,A 0.000,B 0.000,C 90.000,E1 318.038} C_DIS
LIN {X 0.012,Y -378.235,Z 1560.563,A 0.000,B 0.000,C 90.000,E1 317.310} C_DIS
LIN {X 0.002,Y -383.940,Z 1560.531,A 0.000,B 0.000,C 90.000,E1 311.515} C_DIS
LIN {X 0.088,Y -384.893,Z 1560.527,A 0.000,B 0.000,C 90.000,E1 310.782} C_DIS
LIN {X 0.262,Y -390.610,Z 1560.495,A 0.000,B 0.000,C 90.000,E1 305.025} C_DIS
LIN {X 0.106,Y -391.104,Z 1560.493,A 0.000,B 0.000,C 90.000,E1 304.692} C_DIS
LIN {X 0.022,Y -391.648,Z 1560.489,A 0.000,B 0.000,C 90.000,E1 303.992} C_DIS
LIN {X -0.080,Y -396.825,Z 1560.459,A 0.000,B 0.000,C 90.000,E1 298.693} C_DIS
LIN {X -0.210,Y -397.120,Z 1560.457,A 0.000,B 0.000,C 90.000,E1 298.359} C_DIS
LIN {X -0.055,Y -401.597,Z 1560.426,A 0.000,B 0.000,C 90.000,E1 292.717} C_DIS
LIN {X 0.222,Y -404.659,Z 1560.395,A 0.000,B 0.000,C 90.000,E1 287.094} C_DIS
LIN {X -0.079,Y -404.735,Z 1560.391,A 0.000,B 0.000,C 90.000,E1 286.441} C_DIS
LIN {X 0.214,Y -406.099,Z 1560.364,A 0.000,B 0.000,C 90.000,E1 281.535} C_DIS
LIN {X -0.176,Y -406.094,Z 1560.362,A 0.000,B 0.000,C 90.000,E1 281.243} C_DIS
LIN {X -0.097,Y -405.680,Z 1560.333,A 0.000,B 0.000,C 90.000,E1 276.024} C_DIS
LIN {X -0.165,Y -405.058,Z 1560.328,A 0.000,B 0.000,C 90.000,E1 274.992} C_DIS
LIN {X -0.060,Y -403.497,Z 1560.304,A 0.000,B 0.000,C 90.000,E1 270.802} C_DIS
LIN {X -0.092,Y -403.288,Z 1560.302,A 0.000,B 0.000,C 90.000,E1 270.458} C_DIS
LIN {X 0.091,Y -398.931,Z 1560.271,A 0.000,B 0.000,C 90.000,E1 264.837} C_DIS
LIN {X -0.040,Y -393.108,Z 1560.242,A 0.000,B 0.000,C 90.000,E1 259.567} C_DIS
LIN {X -0.079,Y -392.835,Z 1560.240,A 0.000,B 0.000,C 90.000,E1 259.218} C_DIS
LIN {X 0.034,Y -385.993,Z 1560.212,A 0.000,B 0.000,C 90.000,E1 254.212} C_DIS
LIN {X -0.026,Y -385.267,Z 1560.208,A 0.000,B 0.000,C 90.000,E1 253.504} C_DIS
LIN {X -0.004,Y -384.768,Z 1560.206,A 0.000,B 0.000,C 90.000,E1 253.142} C_DIS
LIN {X 0.221,Y -377.973,Z 1560.182,A 0.000,B 0.000,C 90.000,E1 248.773} C_DIS
LIN {X -0.044,Y -376.233,Z 1560.174,A 0.000,B 0.000,C 90.000,E1 247.358} C_DIS
LIN {X 0.057,Y -374.944,Z 1560.170,A 0.000,B 0.000,C 90.000,E1 246.613} C_DIS
LIN {X -0.208,Y -368.417,Z 1560.148,A 0.000,B 0.000,C 90.000,E1 242.615} C_DIS
LIN {X 0.097,Y -366.047,Z 1560.137,A 0.000,B 0.000,C 90.000,E1 240.717} C_DIS
LIN {X 0.004,Y -359.196,Z 1560.115,A 0.000,B 0.000,C 90.000,E1 236.628} C_DIS
LIN {X 0.021,Y -355.842,Z 1560.100,A 0.000,B 0.000,C 90.000,E1 233.989} C_DIS
LIN {X -0.173,Y -348.793,Z 1560.075,A 0.000,B 0.000,C 90.000,E1 229.461} C_DIS
LIN {X -0.097,Y -346.185,Z 1560.062,A 0.000,B 0.000,C 90.000,E1 227.148} C_DIS
LIN {X -0.088,Y -345.065,Z 1560.058,A 0.000,B 0.000,C 90.000,E1 226.377} C_DIS
LIN {X 0.094,Y -338.586,Z 1560.030,A 0.000,B 0.000,C 90.000,E1 221.310} C_DIS
LIN {X 0.094,Y -336.840,Z 1560.019,A 0.000,B 0.000,C 90.000,E1 219.358} C_DIS
LIN {X 0.014,Y -330.861,Z 1559.988,A 0.000,B 0.000,C 90.000,E1 213.865} C_DIS
LIN {X 0.149,Y -329.296,Z 1559.975,A 0.000,B 0.000,C 90.000,E1 211.465} C_DIS
LIN {X -0.154,Y -324.669,Z 1559.942,A 0.000,B 0.000,C 90.000,E1 205.540} C_DIS
LIN {X 0.174,Y -323.837,Z 1559.928,A 0.000,B 0.000,C 90.000,E1 203.078} C_DIS
LIN {X -0.017,Y -321.124,Z 1559.881,A 0.000,B 0.000,C 90.000,E1 194.662} C_DIS
LIN {X 0.138,Y -320.932,Z 1559.877,A 0.000,B 0.000,C 90.000,E1 193.828} C_DIS
LIN {X -0.076,Y -321.562,Z 1559.832,A 0.000,B 0.000,C 90.000,E1 185.796} C_DIS
LIN {X -0.143,Y -324.415,Z 1559.790,A 0.000,B 0.000,C 90.000,E1 178.165} C_DIS
LIN {X -0.141,Y -325.376,Z 1559.783,A 0.000,B 0.000,C 90.000,E1 176.963} C_DIS
LIN {X -0.100,Y -329.112,Z 1559.750,A 0.000,B 0.000,C 90.000,E1 170.971} C_DIS
LIN {X 0.061,Y -334.260,Z 1559.726,A 0.000,B 0.000,C 90.000,E1 166.589} C_DIS
LIN {X 0.067,Y -335.488,Z 1559.719,A 0.000,B 0.000,C 90.000,E1 165.408} C_DIS
LIN {X 0.143,Y -340.932,Z 1559.695,A 0.000,B 0.000,C 90.000,E1 161.094} C_DIS
LIN {X -0.172,Y -342.138,Z 1559.691,A 0.000,B 0.000,C 90.000,E1 160.369} C_DIS
LIN {X -0.058,Y -347.939,Z 1559.667,A 0.000,B 0.000,C 90.000,E1 156.102} C_DIS
LIN {X -0.081,Y -354.259,Z 1559.648,A 0.000,B 0.000,C 90.000,E1 152.666} C_DIS
LIN {X -0.222,Y -361.406,Z 1559.625,A 0.000,B 0.000,C 90.000,E1 148.535} C_DIS
LIN {X 0.065,Y -368.758,Z 1559.606,A 0.000,B 0.000,C 90.000,E1 145.135} C_DIS
LIN {X 0.065,Y -377.029,Z 1559.584,A 0.000,B 0.000,C 90.000,E1 141.090} C_DIS
LIN {X -0.061,Y -383.435,Z 1559.570,A 0.000,B 0.000,C 90.000,E1 138.566} C_DIS
LIN {X -0.015,Y -385.037,Z 1559.566,A 0.000,B 0.000,C 90.000,E1 137.838} C_DIS
LIN {X -0.004,Y -394.325,Z 1559.544,A 0.000,B 0.000,C 90.000,E1 133.905} C_DIS
LIN {X 0.107,Y -399.276,Z 1559.534,A 0.000,B 0.000,C 90.000,E1 132.123} C_DIS
LIN {X 0.210,Y -400.192,Z 1559.532,A 0.000,B 0.000,C 90.000,E1 131.757} C_DIS
LIN {X -0.113,Y -409.687,Z 1559.511,A 0.000,B 0.000,C 90.000,E1 127.971} C_DIS
LIN {X 0.046,Y -415.746,Z 1559.499,A 0.000,B 0.000,C 90.000,E1 125.884} C_DIS
LIN {X 0.153,Y -425.188,Z 1559.479,A 0.000,B 0.000,C 90.000,E1 122.133} C_DIS
LIN {X 0.087,Y -430.186,Z 1559.469,A 0.000,B 0.000,C 90.000,E1 120.463} C_DIS
LIN {X 0.086,Y -431.107,Z 1559.468,A 0.000,B 0.000,C 90.000,E1 120.129} C_DIS
LIN {X -0.129,Y -435.963,Z 1559.456,A 0.000,B 0.000,C 90.000,E1 118.103} C_DIS
LIN {X -0.194,Y -547.819,Z 1559.456,A 0.000,B 0.000,C 90.000,E1 118.103} C_DIS
LIN {X -0.292,Y -548.191,Z 1559.456,A 0.000,B 0.000,C 90.000,E1 118.103} C_DIS
LIN {X -0.308,Y -549.599,Z 1559.455,A 0.000,B 0.000,C 90.000,E1 117.975} C_DIS
LIN {X -0.324,Y -550.357,Z 1559.455,A 0.000,B 0.000,C 90.000,E1 117.847} C_DIS
LIN {X 0.183,Y -551.497,Z 1559.453,A 0.000,B 0.000,C 90.000,E1 117.513} C_DIS
LIN {X -0.281,Y -553.069,Z 1559.450,A 0.000,B 0.000,C 90.000,E1 117.001} C_DIS
LIN {X 0.008,Y -554.189,Z 1559.447,A 0.000,B 0.000,C 90.000,E1 116.411} C_DIS
LIN {X -0.160,Y -555.440,Z 1559.442,A 0.000,B 0.000,C 90.000,E1 115.591} C_DIS
LIN {X 0.194,Y -556.346,Z 1559.438,A 0.000,B 0.000,C 90.000,E1 114.719} C_DIS
LIN {X 0.135,Y -557.323,Z 1559.430,A 0.000,B 0.000,C 90.000,E1 113.334} C_DIS
LIN {X -0.129,Y -557.802,Z 1559.422,A 0.000,B 0.000,C 90.000,E1 111.972} C_DIS
LIN {X 0.133,Y -558.099,Z 1559.414,A 0.000,B 0.000,C 90.000,E1 110.556} C_DIS
LIN {X 0.276,Y -558.388,Z 1559.404,A 0.000,B 0.000,C 90.000,E1 108.598} C_DIS
LIN {X 0.062,Y -558.767,Z 1559.393,A 0.000,B 0.000,C 90.000,E1 106.677} C_DIS
LIN {X -0.035,Y -558.978,Z 1559.385,A 0.000,B 0.000,C 90.000,E1 105.300} C_DIS
LIN {X -0.016,Y -559.158,Z 1559.379,A 0.000,B 0.000,C 90.000,E1 104.189} C_DIS
LIN {X -0.106,Y -559.466,Z 1559.370,A 0.000,B 0.000,C 90.000,E1 102.535} C_DIS
LIN {X -0.174,Y -559.860,Z 1559.359,A 0.000,B 0.000,C 90.000,E1 100.602} C_DIS
LIN {X 0.063,Y -560.386,Z 1559.350,A 0.000,B 0.000,C 90.000,E1 98.916} C_DIS
LIN {X 0.081,Y -560.745,Z 1559.342,A 0.000,B 0.000,C 90.000,E1 97.530} C_DIS
LIN {X -0.226,Y -561.220,Z 1559.331,A 0.000,B 0.000,C 90.000,E1 95.625} C_DIS
LIN {X -0.024,Y -561.731,Z 1559.320,A 0.000,B 0.000,C 90.000,E1 93.669} C_DIS
LIN {X 0.142,Y -562.243,Z 1559.310,A 0.000,B 0.000,C 90.000,E1 91.718} C_DIS
LIN {X -0.275,Y -562.744,Z 1559.299,A 0.000,B 0.000,C 90.000,E1 89.828} C_DIS
LIN {X -0.203,Y -563.222,Z 1559.290,A 0.000,B 0.000,C 90.000,E1 88.165} C_DIS
LIN {X -0.119,Y -563.785,Z 1559.281,A 0.000,B 0.000,C 90.000,E1 86.502} C_DIS
LIN {X 0.004,Y -564.485,Z 1559.271,A 0.000,B 0.000,C 90.000,E1 84.837} C_DIS
LIN {X -0.122,Y -565.555,Z 1559.259,A 0.000,B 0.000,C 90.000,E1 82.648} C_DIS
LIN {X -0.067,Y -566.912,Z 1559.247,A 0.000,B 0.000,C 90.000,E1 80.443} C_DIS
LIN {X -0.248,Y -568.754,Z 1559.233,A 0.000,B 0.000,C 90.000,E1 77.993} C_DIS
LIN {X 0.107,Y -569.820,Z 1559.226,A 0.000,B 0.000,C 90.000,E1 76.589} C_DIS
LIN {X 0.055,Y -570.745,Z 1559.218,A 0.000,B 0.000,C 90.000,E1 75.227} C_DIS
LIN {X 0.168,Y -572.022,Z 1559.206,A 0.000,B 0.000,C 90.000,E1 73.032} C_DIS
LIN {X 0.099,Y -573.262,Z 1559.194,A 0.000,B 0.000,C 90.000,E1 70.859} C_DIS
LIN {X 0.094,Y -574.376,Z 1559.183,A 0.000,B 0.000,C 90.000,E1 68.954} C_DIS
LIN {X 0.120,Y -575.541,Z 1559.173,A 0.000,B 0.000,C 90.000,E1 67.050} C_DIS
LIN {X 0.026,Y -576.261,Z 1559.167,A 0.000,B 0.000,C 90.000,E1 65.973} C_DIS
LIN {X -0.296,Y -576.965,Z 1559.161,A 0.000,B 0.000,C 90.000,E1 64.921} C_DIS
LIN {X -0.183,Y -578.282,Z 1559.149,A 0.000,B 0.000,C 90.000,E1 62.743} C_DIS
LIN {X 0.023,Y -578.897,Z 1559.142,A 0.000,B 0.000,C 90.000,E1 61.641} C_DIS
LIN {X -0.272,Y -579.225,Z 1559.136,A 0.000,B 0.000,C 90.000,E1 60.589} C_DIS
LIN {X 0.083,Y -579.191,Z 1559.132,A 0.000,B 0.000,C 90.000,E1 59.744} C_DIS
LIN {X -0.066,Y -578.831,Z 1559.127,A 0.000,B 0.000,C 90.000,E1 58.948} C_DIS
LIN {X 0.083,Y -578.123,Z 1559.123,A 0.000,B 0.000,C 90.000,E1 58.122} C_DIS
LIN {X -0.072,Y -577.737,Z 1559.121,A 0.000,B 0.000,C 90.000,E1 57.867} C_DIS
LIN {X 0.079,Y -577.159,Z 1559.120,A 0.000,B 0.000,C 90.000,E1 57.582} C_DIS
LIN {X -0.067,Y -576.010,Z 1559.118,A 0.000,B 0.000,C 90.000,E1 57.296} C_DIS
LIN {X 0.158,Y -575.183,Z 1559.118,A 0.000,B 0.000,C 90.000,E1 57.168} C_DIS
LIN {X -0.196,Y -574.514,Z 1559.118,A 0.000,B 0.000,C 90.000,E1 57.168} C_DIS
LIN {X 0.251,Y -574.282,Z 1559.118,A 0.000,B 0.000,C 90.000,E1 57.120} C_DIS
LIN {X 0.168,Y -445.094,Z 1559.118,A 0.000,B 0.000,C 90.000,E1 57.120} C_DIS
LIN {X -0.197,Y -443.714,Z 1559.113,A 0.000,B 0.000,C 90.000,E1 56.421} C_DIS
LIN {X -0.183,Y -434.590,Z 1559.091,A 0.000,B 0.000,C 90.000,E1 52.477} C_DIS
LIN {X -0.070,Y -431.464,Z 1559.082,A 0.000,B 0.000,C 90.000,E1 50.803} C_DIS
LIN {X -0.160,Y -421.581,Z 1559.058,A 0.000,B 0.000,C 90.000,E1 46.458} C_DIS
LIN {X -0.100,Y -418.463,Z 1559.049,A 0.000,B 0.000,C 90.000,E1 44.757} C_DIS
LIN {X -0.012,Y -408.925,Z 1559.024,A 0.000,B 0.000,C 90.000,E1 40.297} C_DIS
LIN {X 0.166,Y -405.999,Z 1559.014,A 0.000,B 0.000,C 90.000,E1 38.543} C_DIS
LIN {X -0.171,Y -397.688,Z 1558.991,A 0.000,B 0.000,C 90.000,E1 34.405} C_DIS
LIN {X -0.089,Y -393.905,Z 1558.977,A 0.000,B 0.000,C 90.000,E1 31.926} C_DIS
LIN {X 0.023,Y -386.494,Z 1558.954,A 0.000,B 0.000,C 90.000,E1 27.641} C_DIS
